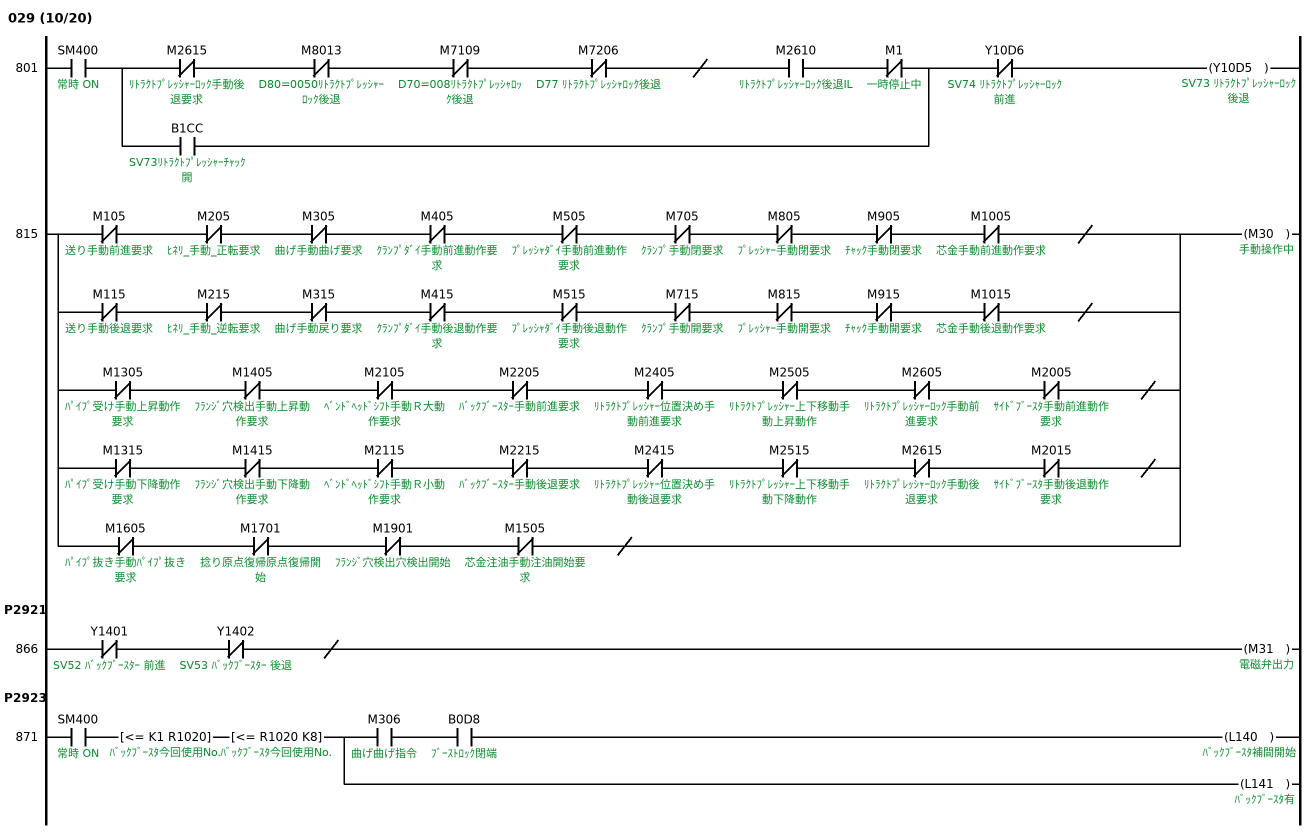
801   LD      SM400  ; 常時 ON
      LDI     M2615  ; ﾘﾄﾗｸﾄﾌﾟﾚｯｼｬｰﾛｯｸ手動後退要求
      ANI     M8013  ; D80=0050ﾘﾄﾗｸﾄﾌﾟﾚｯｼｬｰﾛｯｸ後退
      ANI     M7109  ; D70=008ﾘﾄﾗｸﾄﾌﾟﾚｯｼｬﾛｯｸ後退
      ANI     M7206  ; D77 ﾘﾄﾗｸﾄﾌﾟﾚｯｼｬﾛｯｸ後退
      INV
      AND     M2610  ; ﾘﾄﾗｸﾄﾌﾟﾚｯｼｬｰﾛｯｸ後退IL
      ANI     M1  ; 一時停止中
      OR      B1CC  ; SV73ﾘﾄﾗｸﾄﾌﾟﾚｯｼｬｰﾁｬｯｸ 開
      ANB
      ANI     Y10D6  ; SV74 ﾘﾄﾗｸﾄﾌﾟﾚｯｼｬｰﾛｯｸ 前進
      OUT     Y10D5  ; SV73 ﾘﾄﾗｸﾄﾌﾟﾚｯｼｬｰﾛｯｸ 後退
; 
815   LDI     M105  ; 送り手動前進要求
      ANI     M205  ; ﾋﾈﾘ_手動_正転要求
      ANI     M305  ; 曲げ手動曲げ要求
      ANI     M405  ; ｸﾗﾝﾌﾟﾀﾞｲ手動前進動作要求
      ANI     M505  ; ﾌﾟﾚｯｼｬﾀﾞｲ手動前進動作要求
      ANI     M705  ; ｸﾗﾝﾌﾟ手動閉要求
      ANI     M805  ; ﾌﾟﾚｯｼｬｰ手動閉要求
      ANI     M905  ; ﾁｬｯｸ手動閉要求
      ANI     M1005  ; 芯金手動前進動作要求
      INV
      LDI     M115  ; 送り手動後退要求
      ANI     M215  ; ﾋﾈﾘ_手動_逆転要求
      ANI     M315  ; 曲げ手動戻り要求
      ANI     M415  ; ｸﾗﾝﾌﾟﾀﾞｲ手動後退動作要求
      ANI     M515  ; ﾌﾟﾚｯｼｬﾀﾞｲ手動後退動作要求
      ANI     M715  ; ｸﾗﾝﾌﾟ手動開要求
      ANI     M815  ; ﾌﾟﾚｯｼｬｰ手動開要求
      ANI     M915  ; ﾁｬｯｸ手動開要求
      ANI     M1015  ; 芯金手動後退動作要求
      INV
      ORB
      LDI     M1305  ; ﾊﾟｲﾌﾟ受け手動上昇動作要求
      ANI     M1405  ; ﾌﾗﾝｼﾞ穴検出手動上昇動作要求
      ANI     M2105  ; ﾍﾞﾝﾄﾞﾍｯﾄﾞｼﾌﾄ手動Ｒ大動作要求
      ANI     M2205  ; ﾊﾞｯｸﾌﾞｰｽﾀｰ手動前進要求
      ANI     M2405  ; ﾘﾄﾗｸﾄﾌﾟﾚｯｼｬｰ位置決め手動前進要求
      ANI     M2505  ; ﾘﾄﾗｸﾄﾌﾟﾚｯｼｬｰ上下移動手動上昇動作
      ANI     M2605  ; ﾘﾄﾗｸﾄﾌﾟﾚｯｼｬｰﾛｯｸ手動前進要求
      ANI     M2005  ; ｻｲﾄﾞﾌﾞｰｽﾀ手動前進動作要求
      INV
      ORB
      LDI     M1315  ; ﾊﾟｲﾌﾟ受け手動下降動作要求
      ANI     M1415  ; ﾌﾗﾝｼﾞ穴検出手動下降動作要求
      ANI     M2115  ; ﾍﾞﾝﾄﾞﾍｯﾄﾞｼﾌﾄ手動Ｒ小動作要求
      ANI     M2215  ; ﾊﾞｯｸﾌﾞｰｽﾀｰ手動後退要求
      ANI     M2415  ; ﾘﾄﾗｸﾄﾌﾟﾚｯｼｬｰ位置決め手動後退要求
      ANI     M2515  ; ﾘﾄﾗｸﾄﾌﾟﾚｯｼｬｰ上下移動手動下降動作
      ANI     M2615  ; ﾘﾄﾗｸﾄﾌﾟﾚｯｼｬｰﾛｯｸ手動後退要求
      ANI     M2015  ; ｻｲﾄﾞﾌﾞｰｽﾀ手動後退動作要求
      INV
      ORB
      LDI     M1605  ; ﾊﾟｲﾌﾟ抜き手動ﾊﾟｲﾌﾟ抜き要求
      ANI     M1701  ; 捻り原点復帰原点復帰開始
      ANI     M1901  ; ﾌﾗﾝｼﾞ穴検出穴検出開始
      ANI     M1505  ; 芯金注油手動注油開始要求
      INV
      ORB
      OUT     M30  ; 手動操作中
; 
      P2921
866   LDI     Y1401  ; SV52 ﾊﾞｯｸﾌﾞｰｽﾀｰ 前進
      ANI     Y1402  ; SV53 ﾊﾞｯｸﾌﾞｰｽﾀｰ 後退
      INV
      OUT     M31  ; 電磁弁出力
      P2923
871   LD      SM400  ; 常時 ON
      AND<=   K1 R1020  ; ﾊﾞｯｸﾌﾞｰｽﾀ今回使用No.
      AND<=   R1020 K8  ; ﾊﾞｯｸﾌﾞｰｽﾀ今回使用No.
      MPS
      AND     M306  ; 曲げ曲げ指令
      AND     B0D8  ; ﾌﾞｰｽﾄﾛｯｸ閉端
      OUT     L140  ; ﾊﾞｯｸﾌﾞｰｽﾀ補間開始
      MPP
      OUT     L141  ; ﾊﾞｯｸﾌﾞｰｽﾀ有
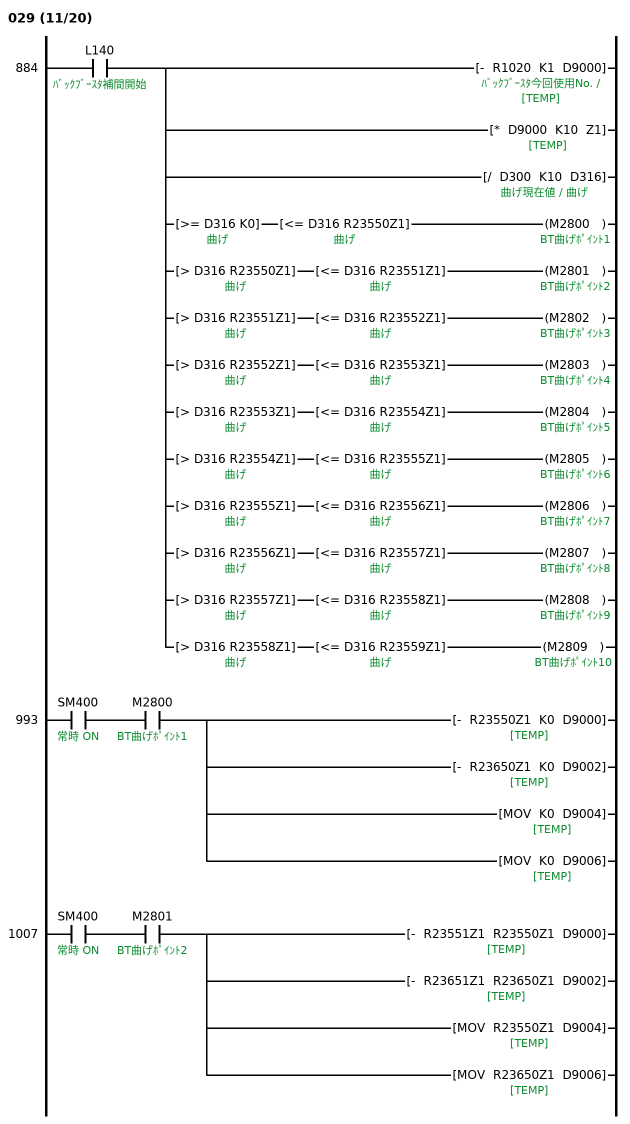
884   LD      L140  ; ﾊﾞｯｸﾌﾞｰｽﾀ補間開始
      -       R1020 K1 D9000  ; [TEMP]
      *       D9000 K10 Z1
      /       D300 K10 D316  ; 曲げ現在値 / 曲げ
      MPS
      AND>=   D316 K0  ; 曲げ
      AND<=   D316 R23550Z1  ; 曲げ
      OUT     M2800  ; BT曲げﾎﾟｲﾝﾄ1
      MRD
      AND>    D316 R23550Z1  ; 曲げ
      AND<=   D316 R23551Z1  ; 曲げ
      OUT     M2801  ; BT曲げﾎﾟｲﾝﾄ2
      MRD
      AND>    D316 R23551Z1  ; 曲げ
      AND<=   D316 R23552Z1  ; 曲げ
      OUT     M2802  ; BT曲げﾎﾟｲﾝﾄ3
      MRD
      AND>    D316 R23552Z1  ; 曲げ
      AND<=   D316 R23553Z1  ; 曲げ
      OUT     M2803  ; BT曲げﾎﾟｲﾝﾄ4
      MRD
      AND>    D316 R23553Z1  ; 曲げ
      AND<=   D316 R23554Z1  ; 曲げ
      OUT     M2804  ; BT曲げﾎﾟｲﾝﾄ5
      MRD
      AND>    D316 R23554Z1  ; 曲げ
      AND<=   D316 R23555Z1  ; 曲げ
      OUT     M2805  ; BT曲げﾎﾟｲﾝﾄ6
      MRD
      AND>    D316 R23555Z1  ; 曲げ
      AND<=   D316 R23556Z1  ; 曲げ
      OUT     M2806  ; BT曲げﾎﾟｲﾝﾄ7
      MRD
      AND>    D316 R23556Z1  ; 曲げ
      AND<=   D316 R23557Z1  ; 曲げ
      OUT     M2807  ; BT曲げﾎﾟｲﾝﾄ8
      MRD
      AND>    D316 R23557Z1  ; 曲げ
      AND<=   D316 R23558Z1  ; 曲げ
      OUT     M2808  ; BT曲げﾎﾟｲﾝﾄ9
      MPP
      AND>    D316 R23558Z1  ; 曲げ
      AND<=   D316 R23559Z1  ; 曲げ
      OUT     M2809  ; BT曲げﾎﾟｲﾝﾄ10
993   LD      SM400  ; 常時 ON
      AND     M2800  ; BT曲げﾎﾟｲﾝﾄ1
      -       R23550Z1 K0 D9000
      -       R23650Z1 K0 D9002  ; [TEMP]
      MOV     K0 D9004  ; [TEMP]
      MOV     K0 D9006  ; [TEMP]
1007  LD      SM400  ; 常時 ON
      AND     M2801  ; BT曲げﾎﾟｲﾝﾄ2
      -       R23551Z1 R23550Z1 D9000
      -       R23651Z1 R23650Z1 D9002
      MOV     R23550Z1 D9004
      MOV     R23650Z1 D9006
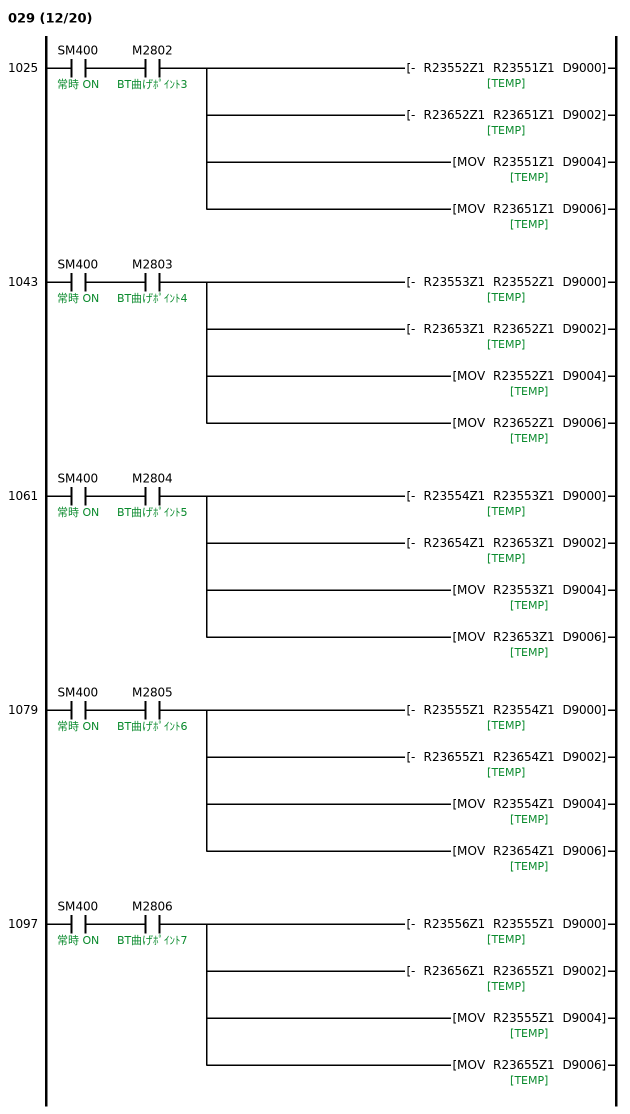
1025  LD      SM400  ; 常時 ON
      AND     M2802  ; BT曲げﾎﾟｲﾝﾄ3
      -       R23552Z1 R23551Z1 D9000
      -       R23652Z1 R23651Z1 D9002
      MOV     R23551Z1 D9004
      MOV     R23651Z1 D9006
1043  LD      SM400  ; 常時 ON
      AND     M2803  ; BT曲げﾎﾟｲﾝﾄ4
      -       R23553Z1 R23552Z1 D9000
      -       R23653Z1 R23652Z1 D9002
      MOV     R23552Z1 D9004
      MOV     R23652Z1 D9006
1061  LD      SM400  ; 常時 ON
      AND     M2804  ; BT曲げﾎﾟｲﾝﾄ5
      -       R23554Z1 R23553Z1 D9000
      -       R23654Z1 R23653Z1 D9002
      MOV     R23553Z1 D9004
      MOV     R23653Z1 D9006
1079  LD      SM400  ; 常時 ON
      AND     M2805  ; BT曲げﾎﾟｲﾝﾄ6
      -       R23555Z1 R23554Z1 D9000
      -       R23655Z1 R23654Z1 D9002
      MOV     R23554Z1 D9004
      MOV     R23654Z1 D9006
1097  LD      SM400  ; 常時 ON
      AND     M2806  ; BT曲げﾎﾟｲﾝﾄ7
      -       R23556Z1 R23555Z1 D9000
      -       R23656Z1 R23655Z1 D9002
      MOV     R23555Z1 D9004
      MOV     R23655Z1 D9006
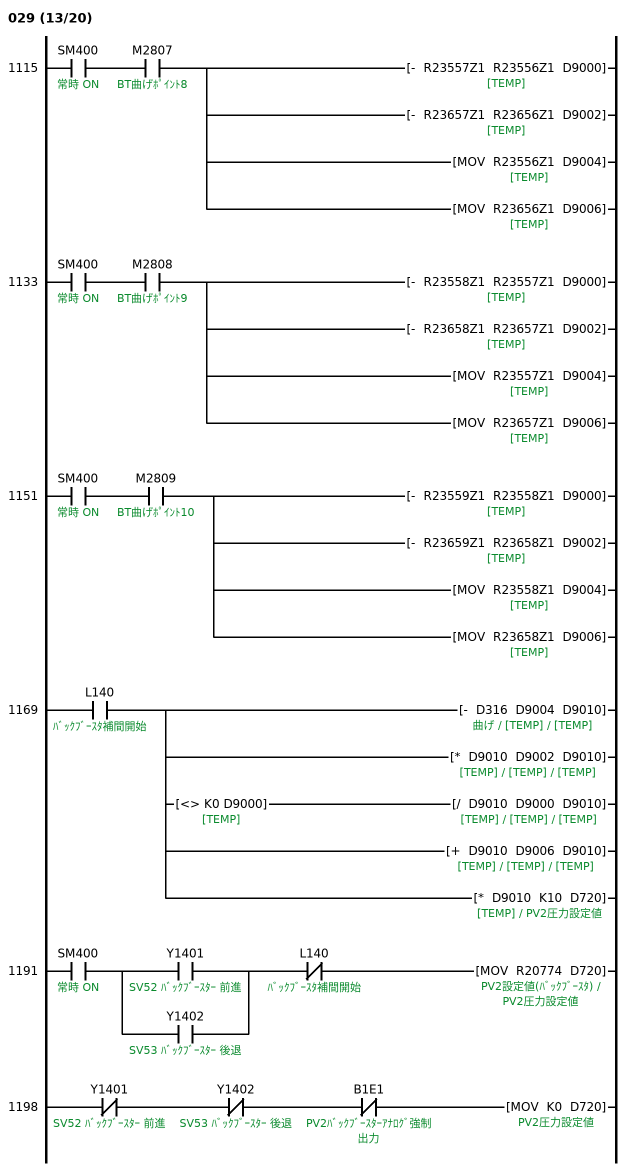
1115  LD      SM400  ; 常時 ON
      AND     M2807  ; BT曲げﾎﾟｲﾝﾄ8
      -       R23557Z1 R23556Z1 D9000
      -       R23657Z1 R23656Z1 D9002
      MOV     R23556Z1 D9004
      MOV     R23656Z1 D9006
1133  LD      SM400  ; 常時 ON
      AND     M2808  ; BT曲げﾎﾟｲﾝﾄ9
      -       R23558Z1 R23557Z1 D9000
      -       R23658Z1 R23657Z1 D9002
      MOV     R23557Z1 D9004
      MOV     R23657Z1 D9006
1151  LD      SM400  ; 常時 ON
      AND     M2809  ; BT曲げﾎﾟｲﾝﾄ10
      -       R23559Z1 R23558Z1 D9000
      -       R23659Z1 R23658Z1 D9002
      MOV     R23558Z1 D9004
      MOV     R23658Z1 D9006
1169  LD      L140  ; ﾊﾞｯｸﾌﾞｰｽﾀ補間開始
      -       D316 D9004 D9010  ; [TEMP]
      *       D9010 D9002 D9010
      MPS
      AND<>   K0 D9000  ; [TEMP]
      /       D9010 D9000 D9010
      MPP
      +       D9010 D9006 D9010
      *       D9010 K10 D720  ; PV2圧力設定値
1191  LD      SM400  ; 常時 ON
      LD      Y1401  ; SV52 ﾊﾞｯｸﾌﾞｰｽﾀｰ 前進
      OR      Y1402  ; SV53 ﾊﾞｯｸﾌﾞｰｽﾀｰ 後退
      ANB
      ANI     L140  ; ﾊﾞｯｸﾌﾞｰｽﾀ補間開始
      MOV     R20774 D720  ; PV2設定値(ﾊﾞｯｸﾌﾞｰｽﾀ)
1198  LDI     Y1401  ; SV52 ﾊﾞｯｸﾌﾞｰｽﾀｰ 前進
      ANI     Y1402  ; SV53 ﾊﾞｯｸﾌﾞｰｽﾀｰ 後退
      ANI     B1E1  ; PV2ﾊﾞｯｸﾌﾞｰｽﾀｰｱﾅﾛｸﾞ強制出力
      MOV     K0 D720
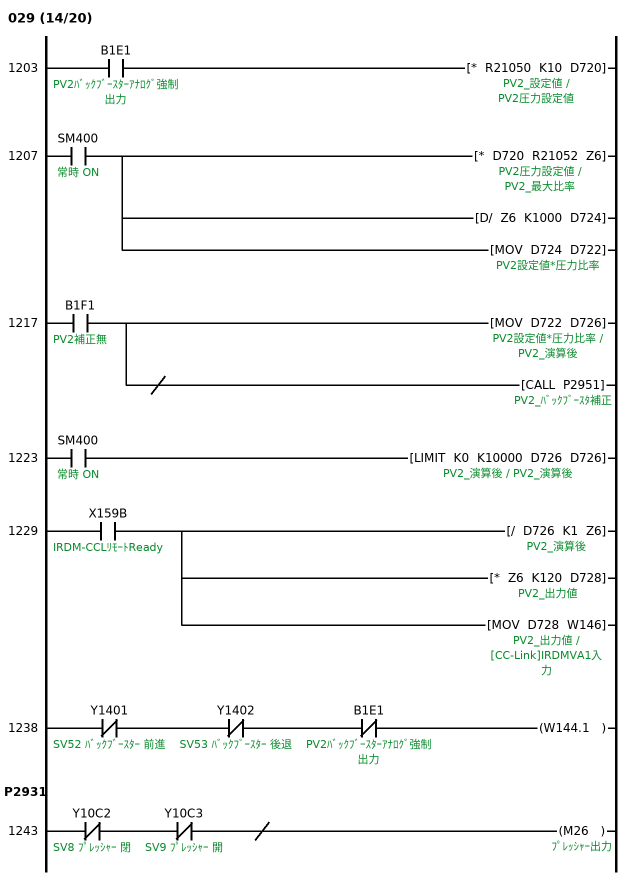
1203  LD      B1E1  ; PV2ﾊﾞｯｸﾌﾞｰｽﾀｰｱﾅﾛｸﾞ強制出力
      *       R21050 K10 D720  ; PV2_設定値
1207  LD      SM400  ; 常時 ON
      *       D720 R21052 Z6  ; PV2_最大比率
      D/      Z6 K1000 D724
      MOV     D724 D722  ; PV2設定値*圧力比率
1217  LD      B1F1  ; PV2補正無
      MOV     D722 D726  ; PV2_演算後
      INV
      CALL    P2951  ; PV2_ﾊﾞｯｸﾌﾞｰｽﾀ補正
1223  LD      SM400  ; 常時 ON
      LIMIT   K0 K10000 D726 D726
1229  LD      X159B  ; IRDM-CCLﾘﾓｰﾄReady
      /       D726 K1 Z6
      *       Z6 K120 D728  ; PV2_出力値
      MOV     D728 W146  ; [CC-Link]IRDMVA1入力
1238  LDI     Y1401  ; SV52 ﾊﾞｯｸﾌﾞｰｽﾀｰ 前進
      ANI     Y1402  ; SV53 ﾊﾞｯｸﾌﾞｰｽﾀｰ 後退
      ANI     B1E1  ; PV2ﾊﾞｯｸﾌﾞｰｽﾀｰｱﾅﾛｸﾞ強制出力
      OUT     W144.1
      P2931
1243  LDI     Y10C2  ; SV8 ﾌﾟﾚｯｼｬｰ 閉
      ANI     Y10C3  ; SV9 ﾌﾟﾚｯｼｬｰ 開
      INV
      OUT     M26  ; ﾌﾟﾚｯｼｬｰ出力
      P2932
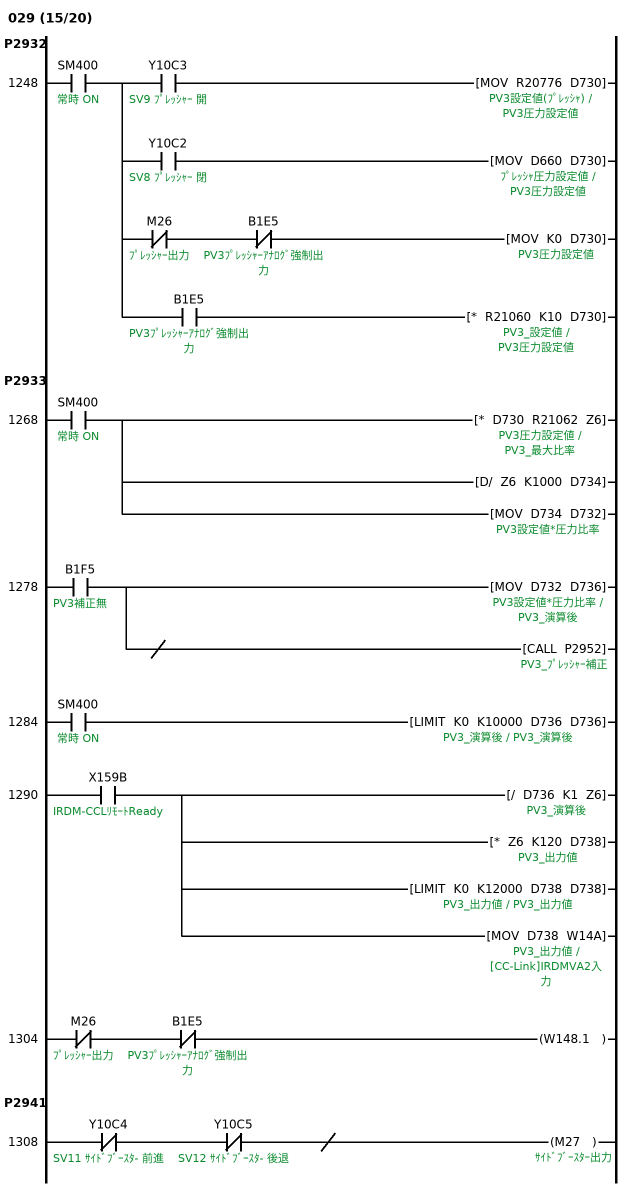
1248  LD      SM400  ; 常時 ON
      MPS
      AND     Y10C3  ; SV9 ﾌﾟﾚｯｼｬｰ 開
      MOV     R20776 D730  ; PV3設定値(ﾌﾟﾚｯｼｬ) / PV3圧力設定値
      MRD
      AND     Y10C2  ; SV8 ﾌﾟﾚｯｼｬｰ 閉
      MOV     D660 D730  ; ﾌﾟﾚｯｼｬ圧力設定値
      MRD
      ANI     M26  ; ﾌﾟﾚｯｼｬｰ出力
      ANI     B1E5  ; PV3ﾌﾟﾚｯｼｬｰｱﾅﾛｸﾞ強制出力
      MOV     K0 D730
      MPP
      AND     B1E5  ; PV3ﾌﾟﾚｯｼｬｰｱﾅﾛｸﾞ強制出力
      *       R21060 K10 D730  ; PV3_設定値
      P2933
1268  LD      SM400  ; 常時 ON
      *       D730 R21062 Z6  ; PV3_最大比率
      D/      Z6 K1000 D734
      MOV     D734 D732  ; PV3設定値*圧力比率
1278  LD      B1F5  ; PV3補正無
      MOV     D732 D736  ; PV3_演算後
      INV
      CALL    P2952  ; PV3_ﾌﾟﾚｯｼｬｰ補正
1284  LD      SM400  ; 常時 ON
      LIMIT   K0 K10000 D736 D736
1290  LD      X159B  ; IRDM-CCLﾘﾓｰﾄReady
      /       D736 K1 Z6
      *       Z6 K120 D738  ; PV3_出力値
      LIMIT   K0 K12000 D738 D738
      MOV     D738 W14A  ; [CC-Link]IRDMVA2入力
1304  LDI     M26  ; ﾌﾟﾚｯｼｬｰ出力
      ANI     B1E5  ; PV3ﾌﾟﾚｯｼｬｰｱﾅﾛｸﾞ強制出力
      OUT     W148.1
      P2941
1308  LDI     Y10C4  ; SV11 ｻｲﾄﾞﾌﾞｰｽﾀ- 前進
      ANI     Y10C5  ; SV12 ｻｲﾄﾞﾌﾞｰｽﾀ- 後退
      INV
      OUT     M27  ; ｻｲﾄﾞﾌﾞｰｽﾀｰ出力
      P2942
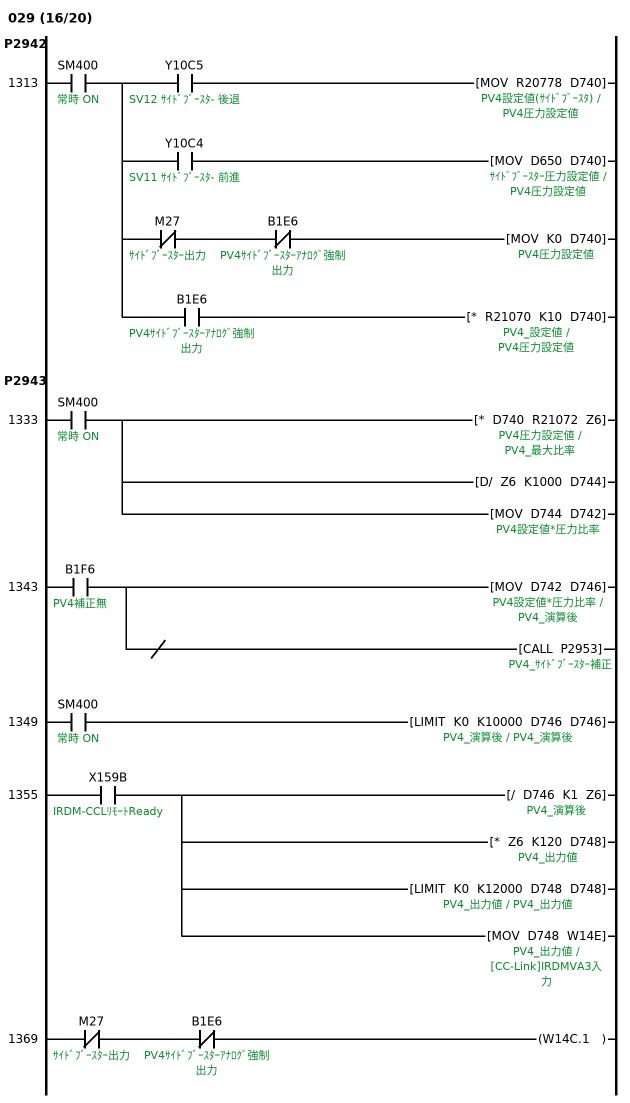
1313  LD      SM400  ; 常時 ON
      MPS
      AND     Y10C5  ; SV12 ｻｲﾄﾞﾌﾞｰｽﾀ- 後退
      MOV     R20778 D740  ; PV4設定値(ｻｲﾄﾞﾌﾞｰｽﾀ) / PV4圧力設定値
      MRD
      AND     Y10C4  ; SV11 ｻｲﾄﾞﾌﾞｰｽﾀ- 前進
      MOV     D650 D740  ; ｻｲﾄﾞﾌﾞｰｽﾀｰ圧力設定値
      MRD
      ANI     M27  ; ｻｲﾄﾞﾌﾞｰｽﾀｰ出力
      ANI     B1E6  ; PV4ｻｲﾄﾞﾌﾞｰｽﾀｰｱﾅﾛｸﾞ強制出力
      MOV     K0 D740
      MPP
      AND     B1E6  ; PV4ｻｲﾄﾞﾌﾞｰｽﾀｰｱﾅﾛｸﾞ強制出力
      *       R21070 K10 D740  ; PV4_設定値
      P2943
1333  LD      SM400  ; 常時 ON
      *       D740 R21072 Z6  ; PV4_最大比率
      D/      Z6 K1000 D744
      MOV     D744 D742  ; PV4設定値*圧力比率
1343  LD      B1F6  ; PV4補正無
      MOV     D742 D746  ; PV4_演算後
      INV
      CALL    P2953  ; PV4_ｻｲﾄﾞﾌﾞｰｽﾀｰ補正
1349  LD      SM400  ; 常時 ON
      LIMIT   K0 K10000 D746 D746
1355  LD      X159B  ; IRDM-CCLﾘﾓｰﾄReady
      /       D746 K1 Z6
      *       Z6 K120 D748  ; PV4_出力値
      LIMIT   K0 K12000 D748 D748
      MOV     D748 W14E  ; [CC-Link]IRDMVA3入力
1369  LDI     M27  ; ｻｲﾄﾞﾌﾞｰｽﾀｰ出力
      ANI     B1E6  ; PV4ｻｲﾄﾞﾌﾞｰｽﾀｰｱﾅﾛｸﾞ強制出力
      OUT     W14C.1
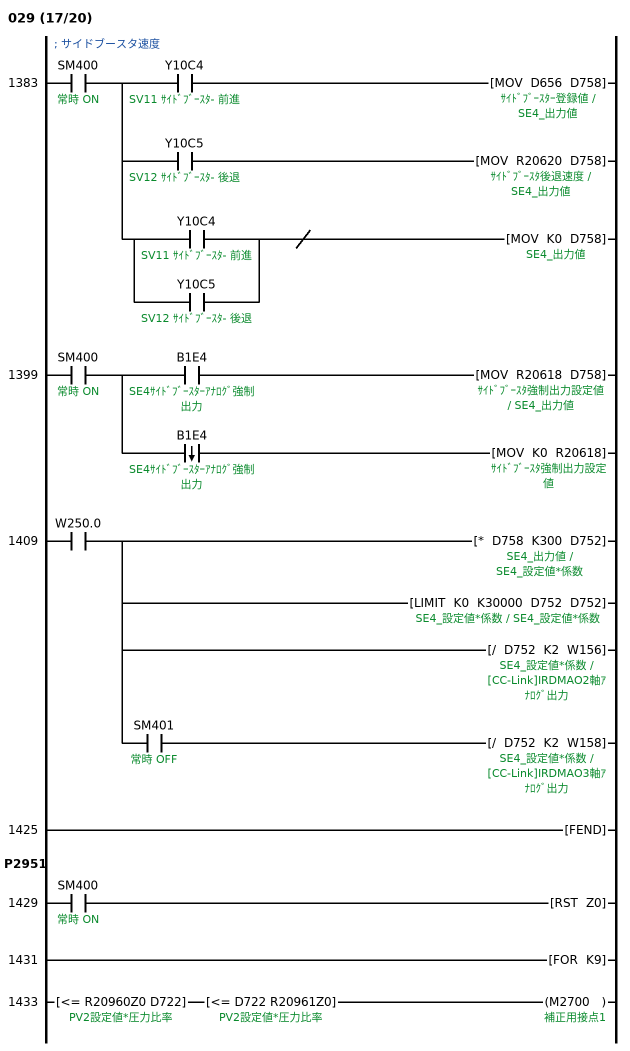
; サイドブースタ速度
1383  LD      SM400  ; 常時 ON
      MPS
      AND     Y10C4  ; SV11 ｻｲﾄﾞﾌﾞｰｽﾀ- 前進
      MOV     D656 D758  ; ｻｲﾄﾞﾌﾞｰｽﾀｰ登録値 / SE4_出力値
      MRD
      AND     Y10C5  ; SV12 ｻｲﾄﾞﾌﾞｰｽﾀ- 後退
      MOV     R20620 D758  ; ｻｲﾄﾞﾌﾞｰｽﾀ後退速度
      MPP
      LD      Y10C4  ; SV11 ｻｲﾄﾞﾌﾞｰｽﾀ- 前進
      OR      Y10C5  ; SV12 ｻｲﾄﾞﾌﾞｰｽﾀ- 後退
      ANB
      INV
      MOV     K0 D758
1399  LD      SM400  ; 常時 ON
      MPS
      AND     B1E4  ; SE4ｻｲﾄﾞﾌﾞｰｽﾀｰｱﾅﾛｸﾞ強制出力
      MOV     R20618 D758  ; ｻｲﾄﾞﾌﾞｰｽﾀ強制出力設定値
      MPP
      ANDF    B1E4  ; SE4ｻｲﾄﾞﾌﾞｰｽﾀｰｱﾅﾛｸﾞ強制出力
      MOV     K0 R20618
1409  LD      W250.0
      *       D758 K300 D752  ; SE4_設定値*係数
      LIMIT   K0 K30000 D752 D752
      /       D752 K2 W156  ; [CC-Link]IRDMAO2軸ｱﾅﾛｸﾞ出力
      AND     SM401  ; 常時 OFF
      /       D752 K2 W158  ; [CC-Link]IRDMAO3軸ｱﾅﾛｸﾞ出力
1425  FEND
; 
      P2951
1429  LD      SM400  ; 常時 ON
      RST     Z0
1431  FOR     K9
1433  LD<=    R20960Z0 D722  ; PV2設定値*圧力比率
      AND<=   D722 R20961Z0  ; PV2設定値*圧力比率
      OUT     M2700  ; 補正用接点1
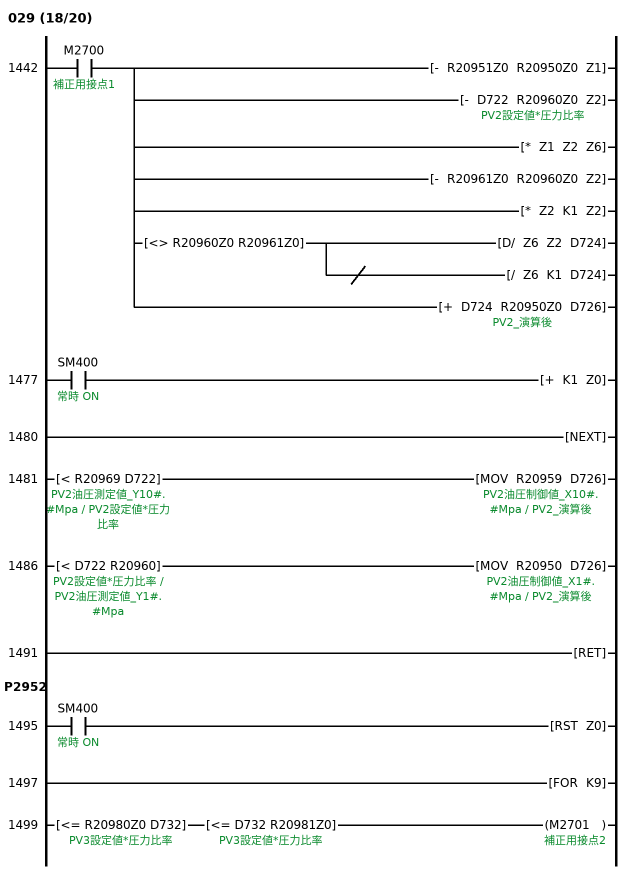
1442  LD      M2700  ; 補正用接点1
      -       R20951Z0 R20950Z0 Z1
      -       D722 R20960Z0 Z2
      *       Z1 Z2 Z6
      -       R20961Z0 R20960Z0 Z2
      *       Z2 K1 Z2
      MPS
      AND<>   R20960Z0 R20961Z0
      D/      Z6 Z2 D724
      INV
      /       Z6 K1 D724
      MPP
      +       D724 R20950Z0 D726
1477  LD      SM400  ; 常時 ON
      +       K1 Z0
1480  NEXT
1481  LD<     R20969 D722  ; PV2油圧測定値_Y10#.#Mpa / PV2設定値*圧力比率
      MOV     R20959 D726  ; PV2油圧制御値_X10#.#Mpa
1486  LD<     D722 R20960  ; PV2設定値*圧力比率 / PV2油圧測定値_Y1#.#Mpa
      MOV     R20950 D726  ; PV2油圧制御値_X1#.#Mpa
1491  RET
; 
      P2952
1495  LD      SM400  ; 常時 ON
      RST     Z0
1497  FOR     K9
1499  LD<=    R20980Z0 D732  ; PV3設定値*圧力比率
      AND<=   D732 R20981Z0  ; PV3設定値*圧力比率
      OUT     M2701  ; 補正用接点2
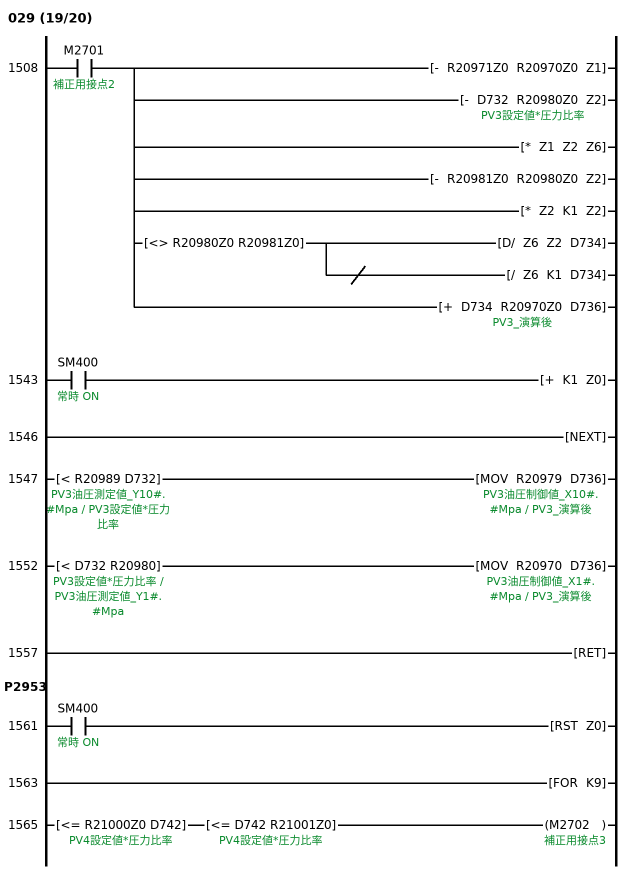
1508  LD      M2701  ; 補正用接点2
      -       R20971Z0 R20970Z0 Z1
      -       D732 R20980Z0 Z2
      *       Z1 Z2 Z6
      -       R20981Z0 R20980Z0 Z2
      *       Z2 K1 Z2
      MPS
      AND<>   R20980Z0 R20981Z0
      D/      Z6 Z2 D734
      INV
      /       Z6 K1 D734
      MPP
      +       D734 R20970Z0 D736
1543  LD      SM400  ; 常時 ON
      +       K1 Z0
1546  NEXT
1547  LD<     R20989 D732  ; PV3油圧測定値_Y10#.#Mpa / PV3設定値*圧力比率
      MOV     R20979 D736  ; PV3油圧制御値_X10#.#Mpa
1552  LD<     D732 R20980  ; PV3設定値*圧力比率 / PV3油圧測定値_Y1#.#Mpa
      MOV     R20970 D736  ; PV3油圧制御値_X1#.#Mpa
1557  RET
; 
      P2953
1561  LD      SM400  ; 常時 ON
      RST     Z0
1563  FOR     K9
1565  LD<=    R21000Z0 D742  ; PV4設定値*圧力比率
      AND<=   D742 R21001Z0  ; PV4設定値*圧力比率
      OUT     M2702  ; 補正用接点3
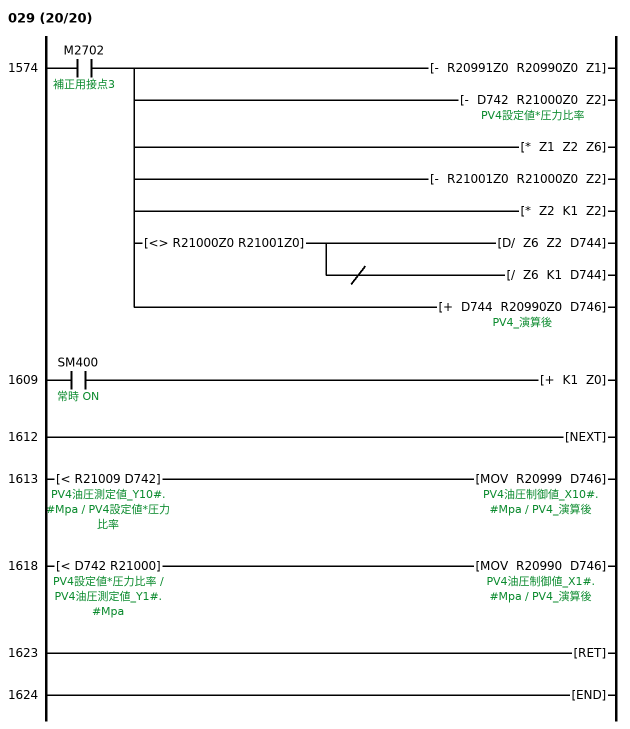
1574  LD      M2702  ; 補正用接点3
      -       R20991Z0 R20990Z0 Z1
      -       D742 R21000Z0 Z2
      *       Z1 Z2 Z6
      -       R21001Z0 R21000Z0 Z2
      *       Z2 K1 Z2
      MPS
      AND<>   R21000Z0 R21001Z0
      D/      Z6 Z2 D744
      INV
      /       Z6 K1 D744
      MPP
      +       D744 R20990Z0 D746
1609  LD      SM400  ; 常時 ON
      +       K1 Z0
1612  NEXT
1613  LD<     R21009 D742  ; PV4油圧測定値_Y10#.#Mpa / PV4設定値*圧力比率
      MOV     R20999 D746  ; PV4油圧制御値_X10#.#Mpa
1618  LD<     D742 R21000  ; PV4設定値*圧力比率 / PV4油圧測定値_Y1#.#Mpa
      MOV     R20990 D746  ; PV4油圧制御値_X1#.#Mpa
1623  RET
1624  END
END_PROGRAM

PROGRAM 030  // TP&表示
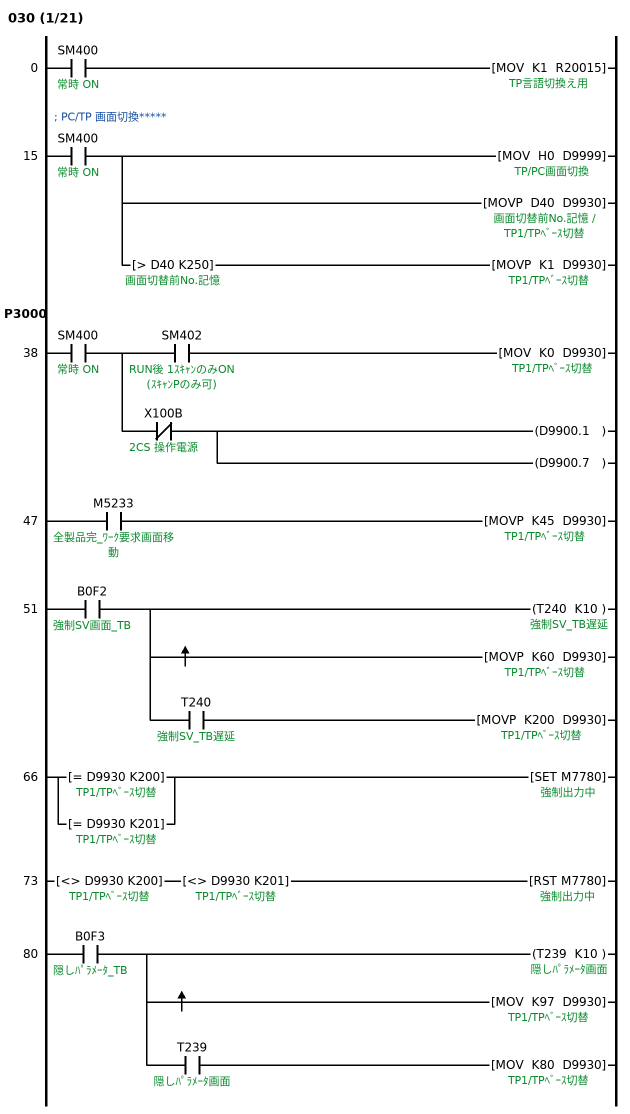
0     LD      SM400  ; 常時 ON
      MOV     K1 R20015  ; TP言語切換え用
; PC/TP 画面切換*****
15    LD      SM400  ; 常時 ON
      MOV     H0 D9999  ; TP/PC画面切換
        [note] ﾀｯﾁﾊﾟﾈﾙ画面
      MOVP    D40 D9930  ; 画面切替前No.記憶 / TP1/TPﾍﾞｰｽ切替
      AND>    D40 K250  ; 画面切替前No.記憶
      MOVP    K1 D9930
; 
      P3000
38    LD      SM400  ; 常時 ON
      MPS
      AND     SM402  ; RUN後 1ｽｷｬﾝのみON (ｽｷｬﾝPのみ可)
      MOV     K0 D9930
      MPP
      ANI     X100B  ; 2CS 操作電源
      OUT     D9900.1
      OUT     D9900.7
47    LD      M5233  ; 全製品完_ﾜｰｸ要求画面移動
      MOVP    K45 D9930
51    LD      B0F2  ; 強制SV画面_TB
      OUT     T240 K10  ; 強制SV_TB遅延
      MPS
      MEP
      MOVP    K60 D9930
      MPP
      AND     T240  ; 強制SV_TB遅延
      MOVP    K200 D9930
66    LD=     D9930 K200  ; TP1/TPﾍﾞｰｽ切替
      OR=     D9930 K201  ; TP1/TPﾍﾞｰｽ切替
      SET     M7780  ; 強制出力中
73    LD<>    D9930 K200  ; TP1/TPﾍﾞｰｽ切替
      AND<>   D9930 K201  ; TP1/TPﾍﾞｰｽ切替
      RST     M7780  ; 強制出力中
80    LD      B0F3  ; 隠しﾊﾟﾗﾒｰﾀ_TB
      OUT     T239 K10  ; 隠しﾊﾟﾗﾒｰﾀ画面
      MPS
      MEP
      MOV     K97 D9930
      MPP
      AND     T239  ; 隠しﾊﾟﾗﾒｰﾀ画面
      MOV     K80 D9930
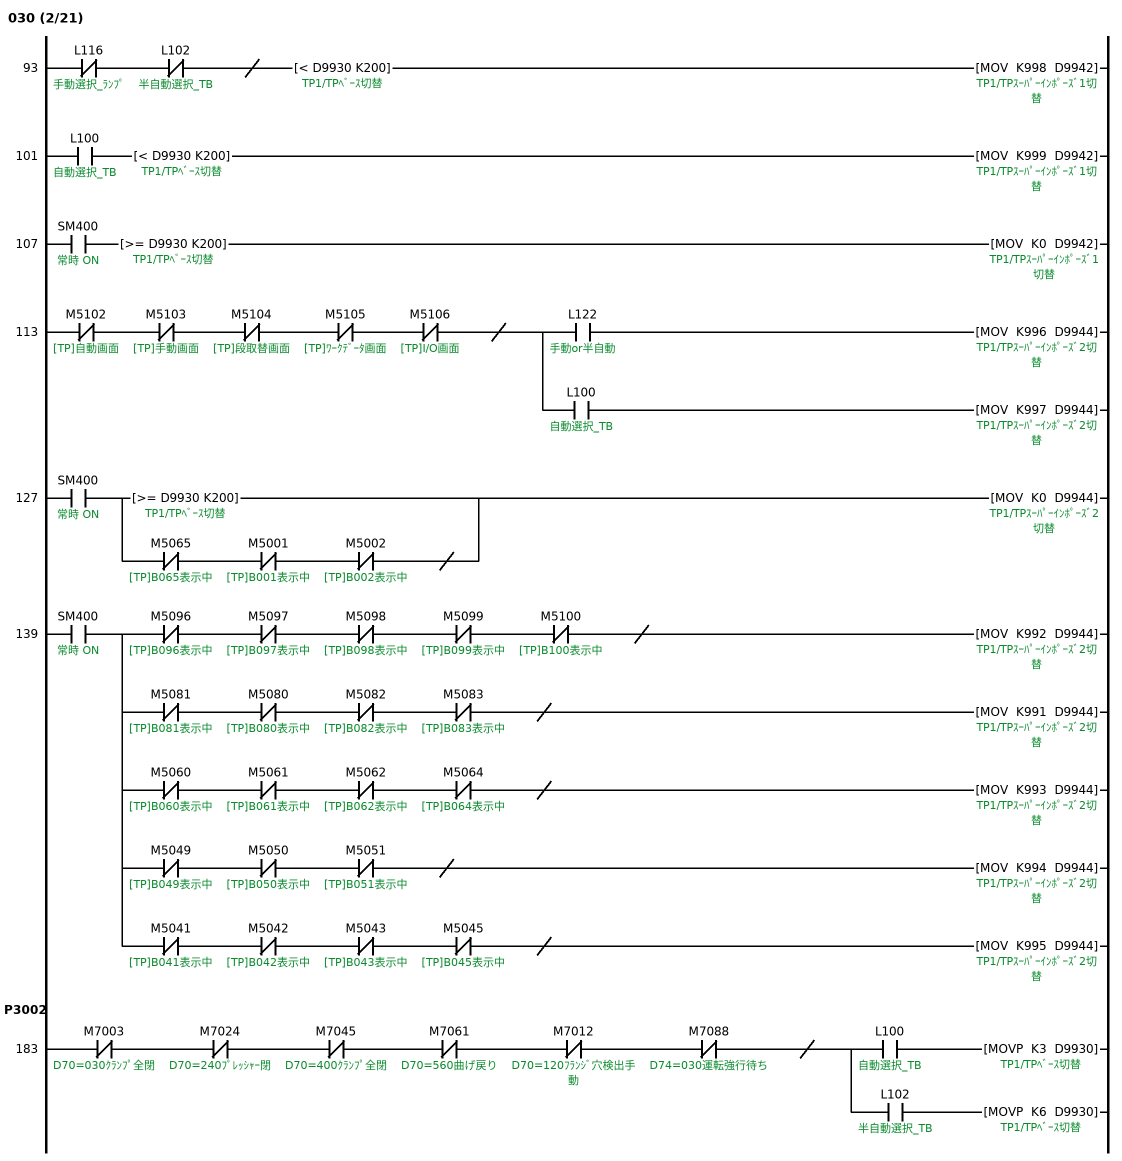
93    LDI     L116  ; 手動選択_ﾗﾝﾌﾟ
      ANI     L102  ; 半自動選択_TB
      INV
      AND<    D9930 K200  ; TP1/TPﾍﾞｰｽ切替
      MOV     K998 D9942  ; TP1/TPｽｰﾊﾟｰｲﾝﾎﾟｰｽﾞ1切替
101   LD      L100  ; 自動選択_TB
      AND<    D9930 K200  ; TP1/TPﾍﾞｰｽ切替
      MOV     K999 D9942
107   LD      SM400  ; 常時 ON
      AND>=   D9930 K200  ; TP1/TPﾍﾞｰｽ切替
      MOV     K0 D9942
113   LDI     M5102  ; [TP]自動画面
      ANI     M5103  ; [TP]手動画面
      ANI     M5104  ; [TP]段取替画面
      ANI     M5105  ; [TP]ﾜｰｸﾃﾞｰﾀ画面
      ANI     M5106  ; [TP]I/O画面
      INV
      MPS
      AND     L122  ; 手動or半自動
      MOV     K996 D9944  ; TP1/TPｽｰﾊﾟｰｲﾝﾎﾟｰｽﾞ2切替
      MPP
      AND     L100  ; 自動選択_TB
      MOV     K997 D9944
127   LD      SM400  ; 常時 ON
      LD>=    D9930 K200  ; TP1/TPﾍﾞｰｽ切替
      LDI     M5065  ; [TP]B065表示中
      ANI     M5001  ; [TP]B001表示中
      ANI     M5002  ; [TP]B002表示中
      INV
      ORB
      ANB
      MOV     K0 D9944
139   LD      SM400  ; 常時 ON
      MPS
      ANI     M5096  ; [TP]B096表示中
      ANI     M5097  ; [TP]B097表示中
      ANI     M5098  ; [TP]B098表示中
      ANI     M5099  ; [TP]B099表示中
      ANI     M5100  ; [TP]B100表示中
      INV
      MOV     K992 D9944
      MRD
      ANI     M5081  ; [TP]B081表示中
      ANI     M5080  ; [TP]B080表示中
      ANI     M5082  ; [TP]B082表示中
      ANI     M5083  ; [TP]B083表示中
      INV
      MOV     K991 D9944
      MRD
      ANI     M5060  ; [TP]B060表示中
      ANI     M5061  ; [TP]B061表示中
      ANI     M5062  ; [TP]B062表示中
      ANI     M5064  ; [TP]B064表示中
      INV
      MOV     K993 D9944
      MRD
      ANI     M5049  ; [TP]B049表示中
      ANI     M5050  ; [TP]B050表示中
      ANI     M5051  ; [TP]B051表示中
      INV
      MOV     K994 D9944
      MPP
      ANI     M5041  ; [TP]B041表示中
      ANI     M5042  ; [TP]B042表示中
      ANI     M5043  ; [TP]B043表示中
      ANI     M5045  ; [TP]B045表示中
      INV
      MOV     K995 D9944
; 
      P3002
183   LDI     M7003  ; D70=030ｸﾗﾝﾌﾟ全閉
      ANI     M7024  ; D70=240ﾌﾟﾚｯｼｬｰ閉
      ANI     M7045  ; D70=400ｸﾗﾝﾌﾟ全閉
      ANI     M7061  ; D70=560曲げ戻り
      ANI     M7012  ; D70=120ﾌﾗﾝｼﾞ穴検出手動
      ANI     M7088  ; D74=030運転強行待ち
      INV
      MPS
      AND     L100  ; 自動選択_TB
      MOVP    K3 D9930
      MPP
      AND     L102  ; 半自動選択_TB
      MOVP    K6 D9930
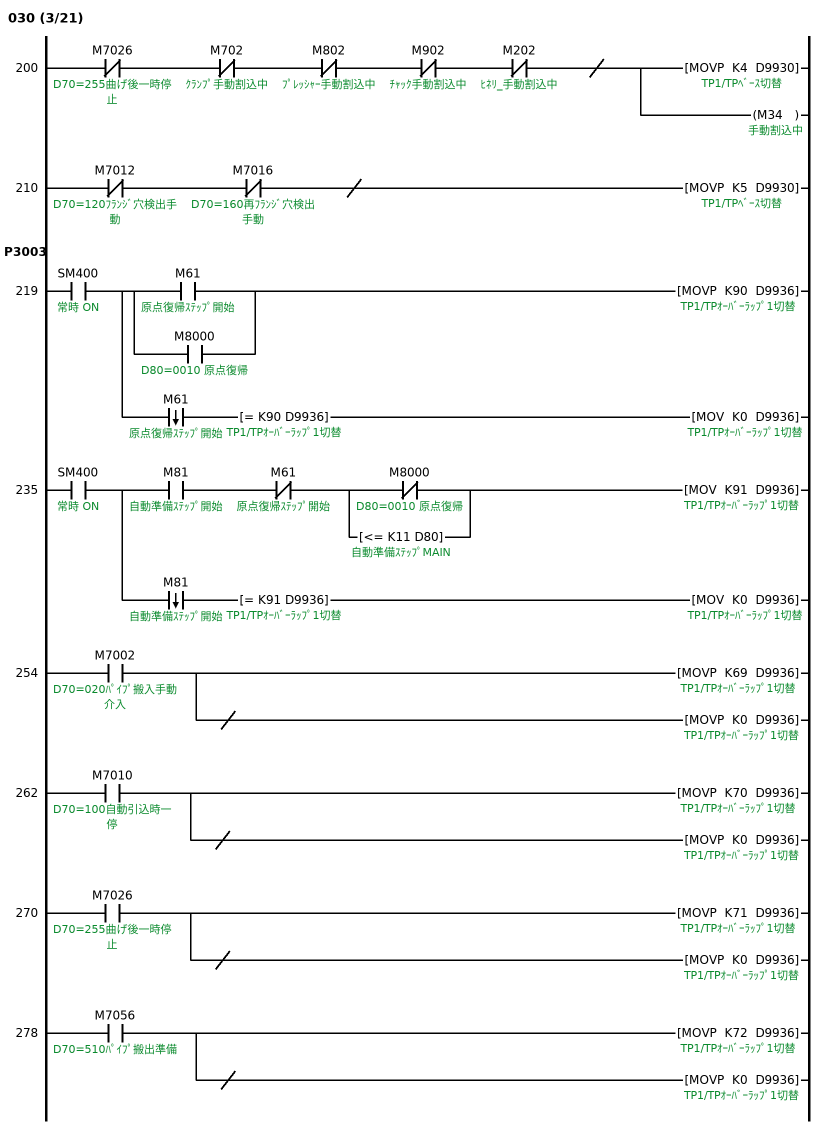
200   LDI     M7026  ; D70=255曲げ後一時停止
      ANI     M702  ; ｸﾗﾝﾌﾟ手動割込中
      ANI     M802  ; ﾌﾟﾚｯｼｬｰ手動割込中
      ANI     M902  ; ﾁｬｯｸ手動割込中
      ANI     M202  ; ﾋﾈﾘ_手動割込中
      INV
      MOVP    K4 D9930
      OUT     M34  ; 手動割込中
210   LDI     M7012  ; D70=120ﾌﾗﾝｼﾞ穴検出手動
      ANI     M7016  ; D70=160再ﾌﾗﾝｼﾞ穴検出手動
      INV
      MOVP    K5 D9930
; 
      P3003
219   LD      SM400  ; 常時 ON
      MPS
      LD      M61  ; 原点復帰ｽﾃｯﾌﾟ開始
      OR      M8000  ; D80=0010 原点復帰
      ANB
      MOVP    K90 D9936  ; TP1/TPｵｰﾊﾞｰﾗｯﾌﾟ1切替
      MPP
      ANDF    M61  ; 原点復帰ｽﾃｯﾌﾟ開始
      AND=    K90 D9936  ; TP1/TPｵｰﾊﾞｰﾗｯﾌﾟ1切替
      MOV     K0 D9936
235   LD      SM400  ; 常時 ON
      MPS
      AND     M81  ; 自動準備ｽﾃｯﾌﾟ開始
      ANI     M61  ; 原点復帰ｽﾃｯﾌﾟ開始
      LDI     M8000  ; D80=0010 原点復帰
      OR<=    K11 D80  ; 自動準備ｽﾃｯﾌﾟMAIN
      ANB
      MOV     K91 D9936
      MPP
      ANDF    M81  ; 自動準備ｽﾃｯﾌﾟ開始
      AND=    K91 D9936  ; TP1/TPｵｰﾊﾞｰﾗｯﾌﾟ1切替
      MOV     K0 D9936
254   LD      M7002  ; D70=020ﾊﾟｲﾌﾟ搬入手動介入
      MOVP    K69 D9936
      INV
      MOVP    K0 D9936
262   LD      M7010  ; D70=100自動引込時一停
      MOVP    K70 D9936
      INV
      MOVP    K0 D9936
270   LD      M7026  ; D70=255曲げ後一時停止
      MOVP    K71 D9936
      INV
      MOVP    K0 D9936
278   LD      M7056  ; D70=510ﾊﾟｲﾌﾟ搬出準備
      MOVP    K72 D9936
      INV
      MOVP    K0 D9936
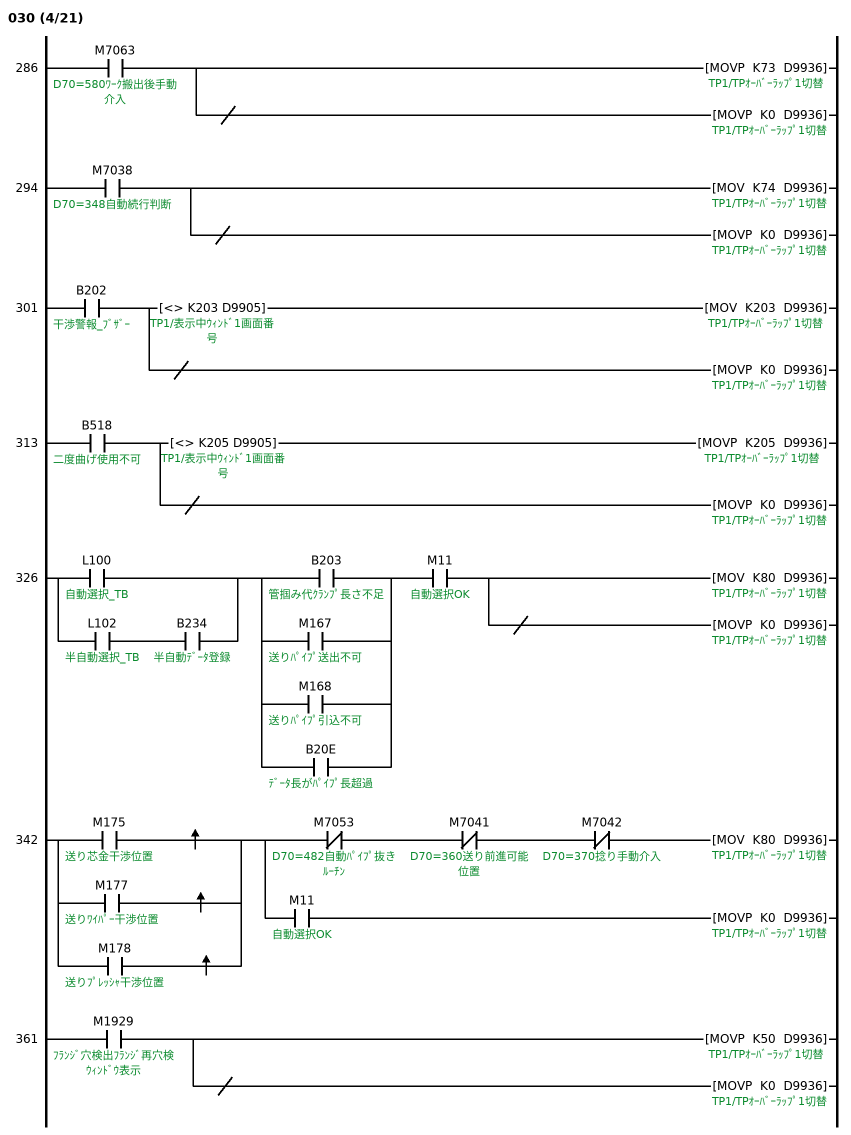
286   LD      M7063  ; D70=580ﾜｰｸ搬出後手動介入
      MOVP    K73 D9936
      INV
      MOVP    K0 D9936
294   LD      M7038  ; D70=348自動続行判断
      MOV     K74 D9936
      INV
      MOVP    K0 D9936
301   LD      B202  ; 干渉警報_ﾌﾞｻﾞｰ
      MPS
      AND<>   K203 D9905  ; TP1/表示中ｳｨﾝﾄﾞ1画面番号
      MOV     K203 D9936
      MPP
      INV
      MOVP    K0 D9936
313   LD      B518  ; 二度曲げ使用不可
      MPS
      AND<>   K205 D9905  ; TP1/表示中ｳｨﾝﾄﾞ1画面番号
      MOVP    K205 D9936
      MPP
      INV
      MOVP    K0 D9936
326   LD      L100  ; 自動選択_TB
      LD      L102  ; 半自動選択_TB
      AND     B234  ; 半自動ﾃﾞｰﾀ登録
      ORB
      LD      B203  ; 管掴み代ｸﾗﾝﾌﾟ長さ不足
      OR      M167  ; 送りﾊﾟｲﾌﾟ送出不可
      OR      M168  ; 送りﾊﾟｲﾌﾟ引込不可
      OR      B20E  ; ﾃﾞｰﾀ長がﾊﾟｲﾌﾟ長超過
      ANB
      AND     M11  ; 自動選択OK
      MOV     K80 D9936
      INV
      MOVP    K0 D9936
342   LD      M175  ; 送り芯金干渉位置
      MEP
      LD      M177  ; 送りﾜｲﾊﾟｰ干渉位置
      MEP
      ORB
      LD      M178  ; 送りﾌﾟﾚｯｼｬ干渉位置
      MEP
      ORB
      MPS
      ANI     M7053  ; D70=482自動ﾊﾟｲﾌﾟ抜きﾙｰﾁﾝ
      ANI     M7041  ; D70=360送り前進可能位置
      ANI     M7042  ; D70=370捻り手動介入
      MOV     K80 D9936
      MPP
      AND     M11  ; 自動選択OK
      MOVP    K0 D9936
361   LD      M1929  ; ﾌﾗﾝｼﾞ穴検出ﾌﾗﾝｼﾞ再穴検ｳｨﾝﾄﾞｳ表示
      MOVP    K50 D9936
      INV
      MOVP    K0 D9936
; 
      P3010
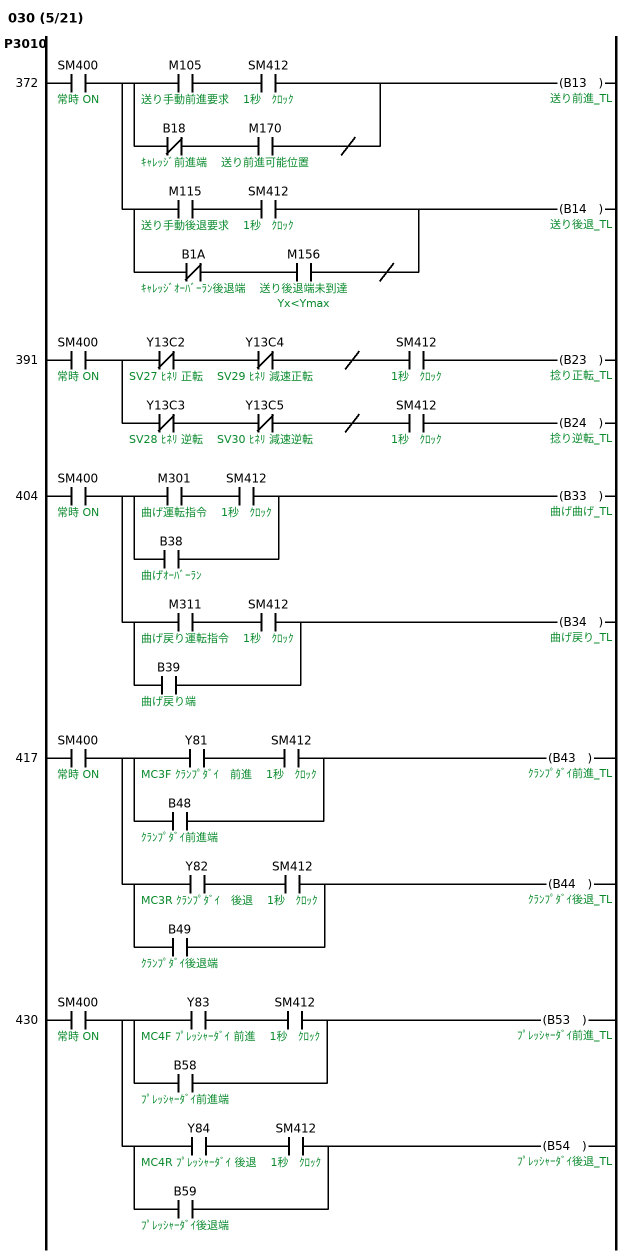
372   LD      SM400  ; 常時 ON
      MPS
      LD      M105  ; 送り手動前進要求
      AND     SM412  ; 1秒   ｸﾛｯｸ
      LDI     B18  ; ｷｬﾚｯｼﾞ前進端
      AND     M170  ; 送り前進可能位置
      INV
      ORB
      ANB
      OUT     B13  ; 送り前進_TL
      MPP
      LD      M115  ; 送り手動後退要求
      AND     SM412  ; 1秒   ｸﾛｯｸ
      LDI     B1A  ; ｷｬﾚｯｼﾞｵｰﾊﾞｰﾗﾝ後退端
      AND     M156  ; 送り後退端未到達 Yx<Ymax
      INV
      ORB
      ANB
      OUT     B14  ; 送り後退_TL
391   LD      SM400  ; 常時 ON
      MPS
      ANI     Y13C2  ; SV27 ﾋﾈﾘ 正転
      ANI     Y13C4  ; SV29 ﾋﾈﾘ 減速正転
      INV
      AND     SM412  ; 1秒   ｸﾛｯｸ
      OUT     B23  ; 捻り正転_TL
      MPP
      ANI     Y13C3  ; SV28 ﾋﾈﾘ 逆転
      ANI     Y13C5  ; SV30 ﾋﾈﾘ 減速逆転
      INV
      AND     SM412  ; 1秒   ｸﾛｯｸ
      OUT     B24  ; 捻り逆転_TL
404   LD      SM400  ; 常時 ON
      MPS
      LD      M301  ; 曲げ運転指令
      AND     SM412  ; 1秒   ｸﾛｯｸ
      OR      B38  ; 曲げｵｰﾊﾞｰﾗﾝ
      ANB
      OUT     B33  ; 曲げ曲げ_TL
      MPP
      LD      M311  ; 曲げ戻り運転指令
      AND     SM412  ; 1秒   ｸﾛｯｸ
      OR      B39  ; 曲げ戻り端
      ANB
      OUT     B34  ; 曲げ戻り_TL
417   LD      SM400  ; 常時 ON
      MPS
      LD      Y81  ; MC3F ｸﾗﾝﾌﾟﾀﾞｲ　前進
      AND     SM412  ; 1秒   ｸﾛｯｸ
      OR      B48  ; ｸﾗﾝﾌﾟﾀﾞｲ前進端
      ANB
      OUT     B43  ; ｸﾗﾝﾌﾟﾀﾞｲ前進_TL
      MPP
      LD      Y82  ; MC3R ｸﾗﾝﾌﾟﾀﾞｲ　後退
      AND     SM412  ; 1秒   ｸﾛｯｸ
      OR      B49  ; ｸﾗﾝﾌﾟﾀﾞｲ後退端
      ANB
      OUT     B44  ; ｸﾗﾝﾌﾟﾀﾞｲ後退_TL
430   LD      SM400  ; 常時 ON
      MPS
      LD      Y83  ; MC4F ﾌﾟﾚｯｼｬｰﾀﾞｲ 前進
      AND     SM412  ; 1秒   ｸﾛｯｸ
      OR      B58  ; ﾌﾟﾚｯｼｬｰﾀﾞｲ前進端
      ANB
      OUT     B53  ; ﾌﾟﾚｯｼｬｰﾀﾞｲ前進_TL
      MPP
      LD      Y84  ; MC4R ﾌﾟﾚｯｼｬｰﾀﾞｲ 後退
      AND     SM412  ; 1秒   ｸﾛｯｸ
      OR      B59  ; ﾌﾟﾚｯｼｬｰﾀﾞｲ後退端
      ANB
      OUT     B54  ; ﾌﾟﾚｯｼｬｰﾀﾞｲ後退_TL
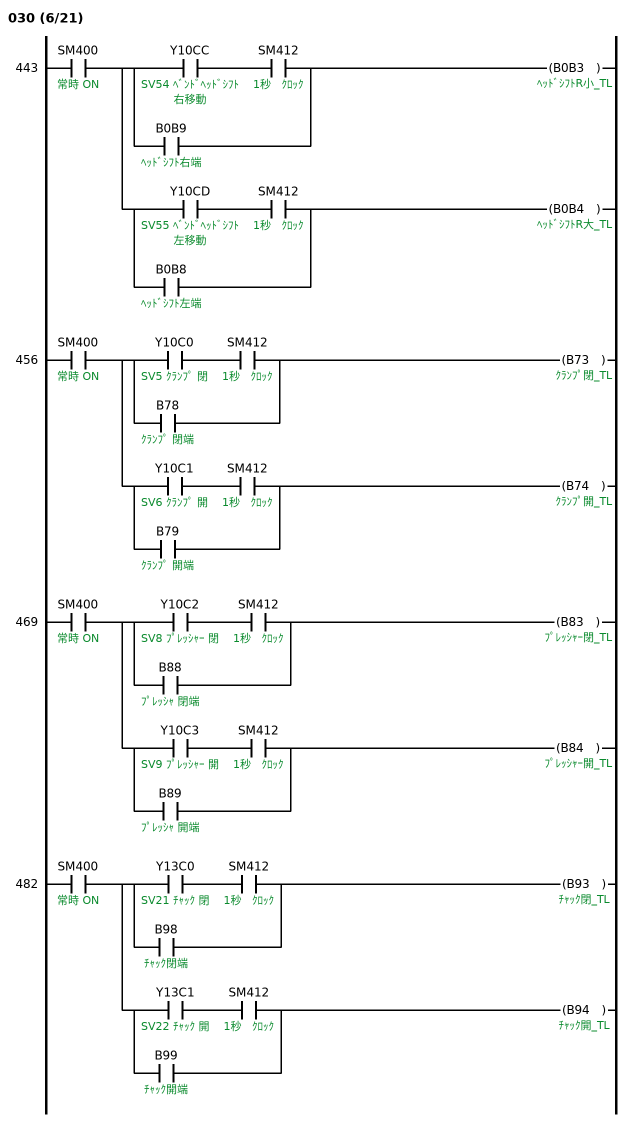
443   LD      SM400  ; 常時 ON
      MPS
      LD      Y10CC  ; SV54 ﾍﾞﾝﾄﾞﾍｯﾄﾞｼﾌﾄ 右移動
      AND     SM412  ; 1秒   ｸﾛｯｸ
      OR      B0B9  ; ﾍｯﾄﾞｼﾌﾄ右端
      ANB
      OUT     B0B3  ; ﾍｯﾄﾞｼﾌﾄR小_TL
      MPP
      LD      Y10CD  ; SV55 ﾍﾞﾝﾄﾞﾍｯﾄﾞｼﾌﾄ 左移動
      AND     SM412  ; 1秒   ｸﾛｯｸ
      OR      B0B8  ; ﾍｯﾄﾞｼﾌﾄ左端
      ANB
      OUT     B0B4  ; ﾍｯﾄﾞｼﾌﾄR大_TL
456   LD      SM400  ; 常時 ON
      MPS
      LD      Y10C0  ; SV5 ｸﾗﾝﾌﾟ 閉
      AND     SM412  ; 1秒   ｸﾛｯｸ
      OR      B78  ; ｸﾗﾝﾌﾟ 閉端
      ANB
      OUT     B73  ; ｸﾗﾝﾌﾟ閉_TL
      MPP
      LD      Y10C1  ; SV6 ｸﾗﾝﾌﾟ 開
      AND     SM412  ; 1秒   ｸﾛｯｸ
      OR      B79  ; ｸﾗﾝﾌﾟ 開端
      ANB
      OUT     B74  ; ｸﾗﾝﾌﾟ開_TL
469   LD      SM400  ; 常時 ON
      MPS
      LD      Y10C2  ; SV8 ﾌﾟﾚｯｼｬｰ 閉
      AND     SM412  ; 1秒   ｸﾛｯｸ
      OR      B88  ; ﾌﾟﾚｯｼｬ 閉端
      ANB
      OUT     B83  ; ﾌﾟﾚｯｼｬｰ閉_TL
      MPP
      LD      Y10C3  ; SV9 ﾌﾟﾚｯｼｬｰ 開
      AND     SM412  ; 1秒   ｸﾛｯｸ
      OR      B89  ; ﾌﾟﾚｯｼｬ 開端
      ANB
      OUT     B84  ; ﾌﾟﾚｯｼｬｰ開_TL
482   LD      SM400  ; 常時 ON
      MPS
      LD      Y13C0  ; SV21 ﾁｬｯｸ 閉
      AND     SM412  ; 1秒   ｸﾛｯｸ
      OR      B98  ; ﾁｬｯｸ閉端
      ANB
      OUT     B93  ; ﾁｬｯｸ閉_TL
      MPP
      LD      Y13C1  ; SV22 ﾁｬｯｸ 開
      AND     SM412  ; 1秒   ｸﾛｯｸ
      OR      B99  ; ﾁｬｯｸ開端
      ANB
      OUT     B94  ; ﾁｬｯｸ開_TL
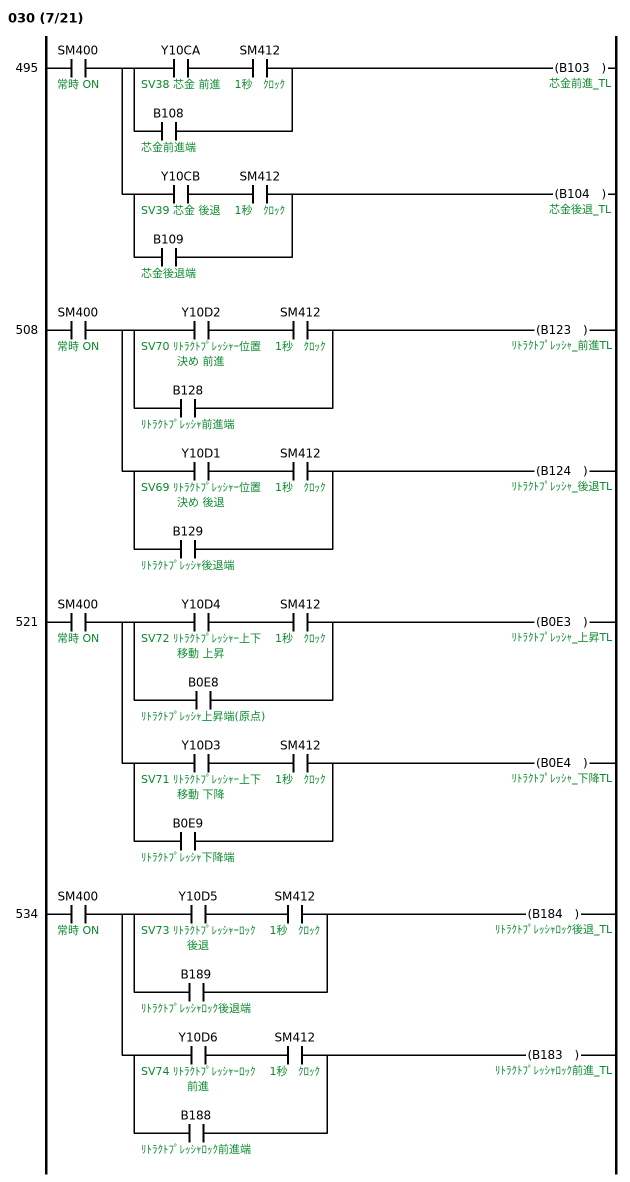
495   LD      SM400  ; 常時 ON
      MPS
      LD      Y10CA  ; SV38 芯金 前進
      AND     SM412  ; 1秒   ｸﾛｯｸ
      OR      B108  ; 芯金前進端
      ANB
      OUT     B103  ; 芯金前進_TL
      MPP
      LD      Y10CB  ; SV39 芯金 後退
      AND     SM412  ; 1秒   ｸﾛｯｸ
      OR      B109  ; 芯金後退端
      ANB
      OUT     B104  ; 芯金後退_TL
508   LD      SM400  ; 常時 ON
      MPS
      LD      Y10D2  ; SV70 ﾘﾄﾗｸﾄﾌﾟﾚｯｼｬｰ位置決め 前進
      AND     SM412  ; 1秒   ｸﾛｯｸ
      OR      B128  ; ﾘﾄﾗｸﾄﾌﾟﾚｯｼｬ前進端
      ANB
      OUT     B123  ; ﾘﾄﾗｸﾄﾌﾟﾚｯｼｬ_前進TL
      MPP
      LD      Y10D1  ; SV69 ﾘﾄﾗｸﾄﾌﾟﾚｯｼｬｰ位置決め 後退
      AND     SM412  ; 1秒   ｸﾛｯｸ
      OR      B129  ; ﾘﾄﾗｸﾄﾌﾟﾚｯｼｬ後退端
      ANB
      OUT     B124  ; ﾘﾄﾗｸﾄﾌﾟﾚｯｼｬ_後退TL
521   LD      SM400  ; 常時 ON
      MPS
      LD      Y10D4  ; SV72 ﾘﾄﾗｸﾄﾌﾟﾚｯｼｬｰ上下移動 上昇
      AND     SM412  ; 1秒   ｸﾛｯｸ
      OR      B0E8  ; ﾘﾄﾗｸﾄﾌﾟﾚｯｼｬ上昇端(原点)
      ANB
      OUT     B0E3  ; ﾘﾄﾗｸﾄﾌﾟﾚｯｼｬ_上昇TL
      MPP
      LD      Y10D3  ; SV71 ﾘﾄﾗｸﾄﾌﾟﾚｯｼｬｰ上下移動 下降
      AND     SM412  ; 1秒   ｸﾛｯｸ
      OR      B0E9  ; ﾘﾄﾗｸﾄﾌﾟﾚｯｼｬ下降端
      ANB
      OUT     B0E4  ; ﾘﾄﾗｸﾄﾌﾟﾚｯｼｬ_下降TL
534   LD      SM400  ; 常時 ON
      MPS
      LD      Y10D5  ; SV73 ﾘﾄﾗｸﾄﾌﾟﾚｯｼｬｰﾛｯｸ 後退
      AND     SM412  ; 1秒   ｸﾛｯｸ
      OR      B189  ; ﾘﾄﾗｸﾄﾌﾟﾚｯｼｬﾛｯｸ後退端
      ANB
      OUT     B184  ; ﾘﾄﾗｸﾄﾌﾟﾚｯｼｬﾛｯｸ後退_TL
      MPP
      LD      Y10D6  ; SV74 ﾘﾄﾗｸﾄﾌﾟﾚｯｼｬｰﾛｯｸ 前進
      AND     SM412  ; 1秒   ｸﾛｯｸ
      OR      B188  ; ﾘﾄﾗｸﾄﾌﾟﾚｯｼｬﾛｯｸ前進端
      ANB
      OUT     B183  ; ﾘﾄﾗｸﾄﾌﾟﾚｯｼｬﾛｯｸ前進_TL
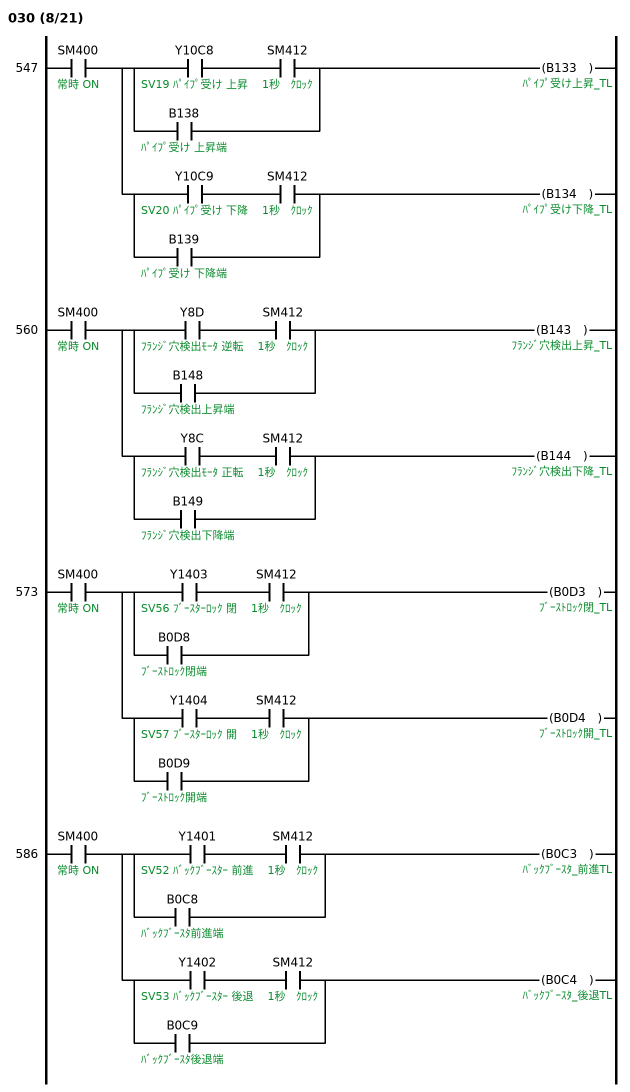
547   LD      SM400  ; 常時 ON
      MPS
      LD      Y10C8  ; SV19 ﾊﾟｲﾌﾟ受け 上昇
      AND     SM412  ; 1秒   ｸﾛｯｸ
      OR      B138  ; ﾊﾟｲﾌﾟ受け 上昇端
      ANB
      OUT     B133  ; ﾊﾟｲﾌﾟ受け上昇_TL
      MPP
      LD      Y10C9  ; SV20 ﾊﾟｲﾌﾟ受け 下降
      AND     SM412  ; 1秒   ｸﾛｯｸ
      OR      B139  ; ﾊﾟｲﾌﾟ受け 下降端
      ANB
      OUT     B134  ; ﾊﾟｲﾌﾟ受け下降_TL
560   LD      SM400  ; 常時 ON
      MPS
      LD      Y8D  ; ﾌﾗﾝｼﾞ穴検出ﾓｰﾀ 逆転
      AND     SM412  ; 1秒   ｸﾛｯｸ
      OR      B148  ; ﾌﾗﾝｼﾞ穴検出上昇端
      ANB
      OUT     B143  ; ﾌﾗﾝｼﾞ穴検出上昇_TL
      MPP
      LD      Y8C  ; ﾌﾗﾝｼﾞ穴検出ﾓｰﾀ 正転
      AND     SM412  ; 1秒   ｸﾛｯｸ
      OR      B149  ; ﾌﾗﾝｼﾞ穴検出下降端
      ANB
      OUT     B144  ; ﾌﾗﾝｼﾞ穴検出下降_TL
573   LD      SM400  ; 常時 ON
      MPS
      LD      Y1403  ; SV56 ﾌﾞｰｽﾀｰﾛｯｸ 閉
      AND     SM412  ; 1秒   ｸﾛｯｸ
      OR      B0D8  ; ﾌﾞｰｽﾄﾛｯｸ閉端
      ANB
      OUT     B0D3  ; ﾌﾞｰｽﾄﾛｯｸ閉_TL
      MPP
      LD      Y1404  ; SV57 ﾌﾞｰｽﾀｰﾛｯｸ 開
      AND     SM412  ; 1秒   ｸﾛｯｸ
      OR      B0D9  ; ﾌﾞｰｽﾄﾛｯｸ開端
      ANB
      OUT     B0D4  ; ﾌﾞｰｽﾄﾛｯｸ開_TL
586   LD      SM400  ; 常時 ON
      MPS
      LD      Y1401  ; SV52 ﾊﾞｯｸﾌﾞｰｽﾀｰ 前進
      AND     SM412  ; 1秒   ｸﾛｯｸ
      OR      B0C8  ; ﾊﾞｯｸﾌﾞｰｽﾀ前進端
      ANB
      OUT     B0C3  ; ﾊﾞｯｸﾌﾞｰｽﾀ_前進TL
      MPP
      LD      Y1402  ; SV53 ﾊﾞｯｸﾌﾞｰｽﾀｰ 後退
      AND     SM412  ; 1秒   ｸﾛｯｸ
      OR      B0C9  ; ﾊﾞｯｸﾌﾞｰｽﾀ後退端
      ANB
      OUT     B0C4  ; ﾊﾞｯｸﾌﾞｰｽﾀ_後退TL
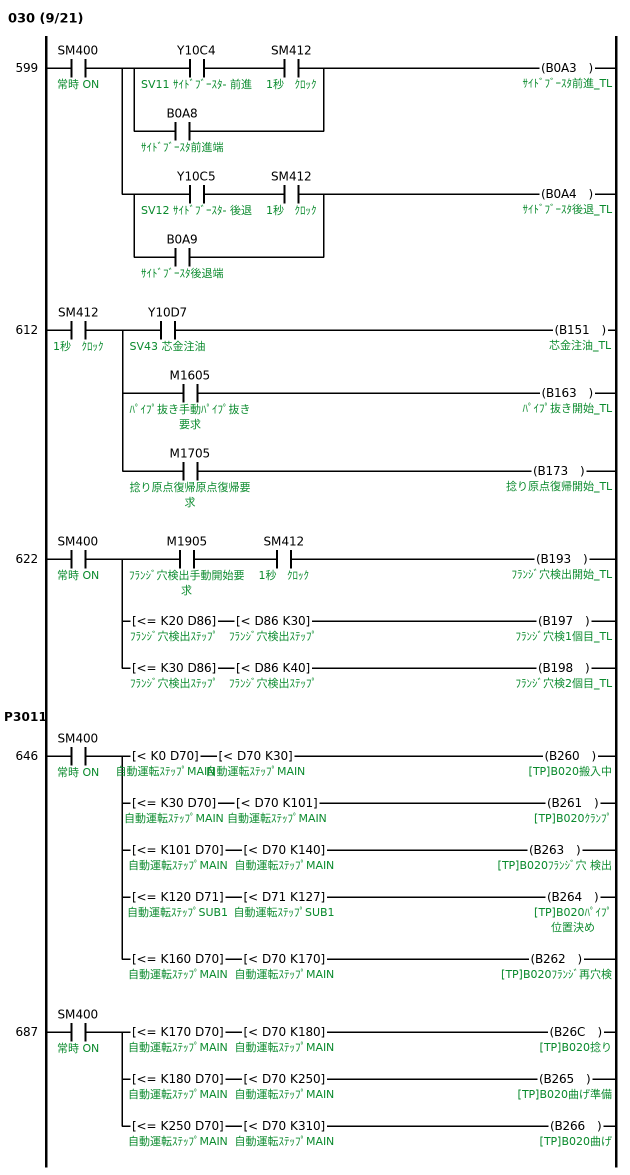
599   LD      SM400  ; 常時 ON
      MPS
      LD      Y10C4  ; SV11 ｻｲﾄﾞﾌﾞｰｽﾀ- 前進
      AND     SM412  ; 1秒   ｸﾛｯｸ
      OR      B0A8  ; ｻｲﾄﾞﾌﾞｰｽﾀ前進端
      ANB
      OUT     B0A3  ; ｻｲﾄﾞﾌﾞｰｽﾀ前進_TL
      MPP
      LD      Y10C5  ; SV12 ｻｲﾄﾞﾌﾞｰｽﾀ- 後退
      AND     SM412  ; 1秒   ｸﾛｯｸ
      OR      B0A9  ; ｻｲﾄﾞﾌﾞｰｽﾀ後退端
      ANB
      OUT     B0A4  ; ｻｲﾄﾞﾌﾞｰｽﾀ後退_TL
612   LD      SM412  ; 1秒   ｸﾛｯｸ
      MPS
      AND     Y10D7  ; SV43 芯金注油
      OUT     B151  ; 芯金注油_TL
      MRD
      AND     M1605  ; ﾊﾟｲﾌﾟ抜き手動ﾊﾟｲﾌﾟ抜き要求
      OUT     B163  ; ﾊﾟｲﾌﾟ抜き開始_TL
      MPP
      AND     M1705  ; 捻り原点復帰原点復帰要求
      OUT     B173  ; 捻り原点復帰開始_TL
622   LD      SM400  ; 常時 ON
      MPS
      AND     M1905  ; ﾌﾗﾝｼﾞ穴検出手動開始要求
      AND     SM412  ; 1秒   ｸﾛｯｸ
      OUT     B193  ; ﾌﾗﾝｼﾞ穴検出開始_TL
      MRD
      AND<=   K20 D86  ; ﾌﾗﾝｼﾞ穴検出ｽﾃｯﾌﾟ
      AND<    D86 K30  ; ﾌﾗﾝｼﾞ穴検出ｽﾃｯﾌﾟ
      OUT     B197  ; ﾌﾗﾝｼﾞ穴検1個目_TL
      MPP
      AND<=   K30 D86  ; ﾌﾗﾝｼﾞ穴検出ｽﾃｯﾌﾟ
      AND<    D86 K40  ; ﾌﾗﾝｼﾞ穴検出ｽﾃｯﾌﾟ
      OUT     B198  ; ﾌﾗﾝｼﾞ穴検2個目_TL
; 
      P3011
646   LD      SM400  ; 常時 ON
      MPS
      AND<    K0 D70  ; 自動運転ｽﾃｯﾌﾟMAIN
      AND<    D70 K30  ; 自動運転ｽﾃｯﾌﾟMAIN
      OUT     B260  ; [TP]B020搬入中
      MRD
      AND<=   K30 D70  ; 自動運転ｽﾃｯﾌﾟMAIN
      AND<    D70 K101  ; 自動運転ｽﾃｯﾌﾟMAIN
      OUT     B261  ; [TP]B020ｸﾗﾝﾌﾟ
      MRD
      AND<=   K101 D70  ; 自動運転ｽﾃｯﾌﾟMAIN
      AND<    D70 K140  ; 自動運転ｽﾃｯﾌﾟMAIN
      OUT     B263  ; [TP]B020ﾌﾗﾝｼﾞ穴 検出
      MRD
      AND<=   K120 D71  ; 自動運転ｽﾃｯﾌﾟSUB1
      AND<    D71 K127  ; 自動運転ｽﾃｯﾌﾟSUB1
      OUT     B264  ; [TP]B020ﾊﾟｲﾌﾟ   位置決め
      MPP
      AND<=   K160 D70  ; 自動運転ｽﾃｯﾌﾟMAIN
      AND<    D70 K170  ; 自動運転ｽﾃｯﾌﾟMAIN
      OUT     B262  ; [TP]B020ﾌﾗﾝｼﾞ再穴検
687   LD      SM400  ; 常時 ON
      MPS
      AND<=   K170 D70  ; 自動運転ｽﾃｯﾌﾟMAIN
      AND<    D70 K180  ; 自動運転ｽﾃｯﾌﾟMAIN
      OUT     B26C  ; [TP]B020捻り
      MRD
      AND<=   K180 D70  ; 自動運転ｽﾃｯﾌﾟMAIN
      AND<    D70 K250  ; 自動運転ｽﾃｯﾌﾟMAIN
      OUT     B265  ; [TP]B020曲げ準備
      MPP
      AND<=   K250 D70  ; 自動運転ｽﾃｯﾌﾟMAIN
      AND<    D70 K310  ; 自動運転ｽﾃｯﾌﾟMAIN
      OUT     B266  ; [TP]B020曲げ
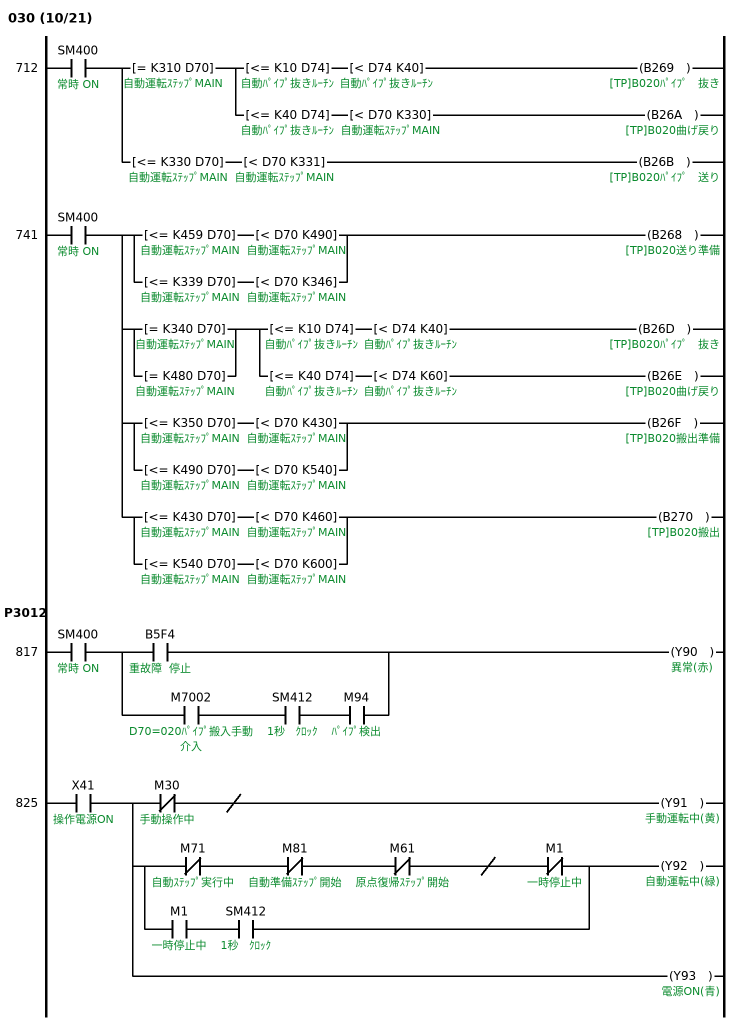
712   LD      SM400  ; 常時 ON
      MPS
      AND=    K310 D70  ; 自動運転ｽﾃｯﾌﾟMAIN
      MPS
      AND<=   K10 D74  ; 自動ﾊﾟｲﾌﾟ抜きﾙｰﾁﾝ
      AND<    D74 K40  ; 自動ﾊﾟｲﾌﾟ抜きﾙｰﾁﾝ
      OUT     B269  ; [TP]B020ﾊﾟｲﾌﾟ   抜き
      MPP
      AND<=   K40 D74  ; 自動ﾊﾟｲﾌﾟ抜きﾙｰﾁﾝ
      AND<    D70 K330  ; 自動運転ｽﾃｯﾌﾟMAIN
      OUT     B26A  ; [TP]B020曲げ戻り
      MPP
      AND<=   K330 D70  ; 自動運転ｽﾃｯﾌﾟMAIN
      AND<    D70 K331  ; 自動運転ｽﾃｯﾌﾟMAIN
      OUT     B26B  ; [TP]B020ﾊﾟｲﾌﾟ   送り
741   LD      SM400  ; 常時 ON
      MPS
      LD<=    K459 D70  ; 自動運転ｽﾃｯﾌﾟMAIN
      AND<    D70 K490  ; 自動運転ｽﾃｯﾌﾟMAIN
      LD<=    K339 D70  ; 自動運転ｽﾃｯﾌﾟMAIN
      AND<    D70 K346  ; 自動運転ｽﾃｯﾌﾟMAIN
      ORB
      ANB
      OUT     B268  ; [TP]B020送り準備
      MRD
      LD=     K340 D70  ; 自動運転ｽﾃｯﾌﾟMAIN
      OR=     K480 D70  ; 自動運転ｽﾃｯﾌﾟMAIN
      ANB
      MPS
      AND<=   K10 D74  ; 自動ﾊﾟｲﾌﾟ抜きﾙｰﾁﾝ
      AND<    D74 K40  ; 自動ﾊﾟｲﾌﾟ抜きﾙｰﾁﾝ
      OUT     B26D  ; [TP]B020ﾊﾟｲﾌﾟ   抜き
      MPP
      AND<=   K40 D74  ; 自動ﾊﾟｲﾌﾟ抜きﾙｰﾁﾝ
      AND<    D74 K60  ; 自動ﾊﾟｲﾌﾟ抜きﾙｰﾁﾝ
      OUT     B26E  ; [TP]B020曲げ戻り
      MRD
      LD<=    K350 D70  ; 自動運転ｽﾃｯﾌﾟMAIN
      AND<    D70 K430  ; 自動運転ｽﾃｯﾌﾟMAIN
      LD<=    K490 D70  ; 自動運転ｽﾃｯﾌﾟMAIN
      AND<    D70 K540  ; 自動運転ｽﾃｯﾌﾟMAIN
      ORB
      ANB
      OUT     B26F  ; [TP]B020搬出準備
      MPP
      LD<=    K430 D70  ; 自動運転ｽﾃｯﾌﾟMAIN
      AND<    D70 K460  ; 自動運転ｽﾃｯﾌﾟMAIN
      LD<=    K540 D70  ; 自動運転ｽﾃｯﾌﾟMAIN
      AND<    D70 K600  ; 自動運転ｽﾃｯﾌﾟMAIN
      ORB
      ANB
      OUT     B270  ; [TP]B020搬出
; 
      P3012
817   LD      SM400  ; 常時 ON
      LD      B5F4  ; 重故障  停止
      LD      M7002  ; D70=020ﾊﾟｲﾌﾟ搬入手動介入
      AND     SM412  ; 1秒   ｸﾛｯｸ
      AND     M94  ; ﾊﾟｲﾌﾟ検出
      ORB
      ANB
      OUT     Y90  ; 異常(赤)
825   LD      X41  ; 操作電源ON
      MPS
      ANI     M30  ; 手動操作中
      INV
      OUT     Y91  ; 手動運転中(黄)
      MRD
      LDI     M71  ; 自動ｽﾃｯﾌﾟ実行中
      ANI     M81  ; 自動準備ｽﾃｯﾌﾟ開始
      ANI     M61  ; 原点復帰ｽﾃｯﾌﾟ開始
      INV
      ANI     M1  ; 一時停止中
      LD      M1  ; 一時停止中
      AND     SM412  ; 1秒   ｸﾛｯｸ
      ORB
      ANB
      OUT     Y92  ; 自動運転中(緑)
      MPP
      OUT     Y93  ; 電源ON(青)
; 
      P3013
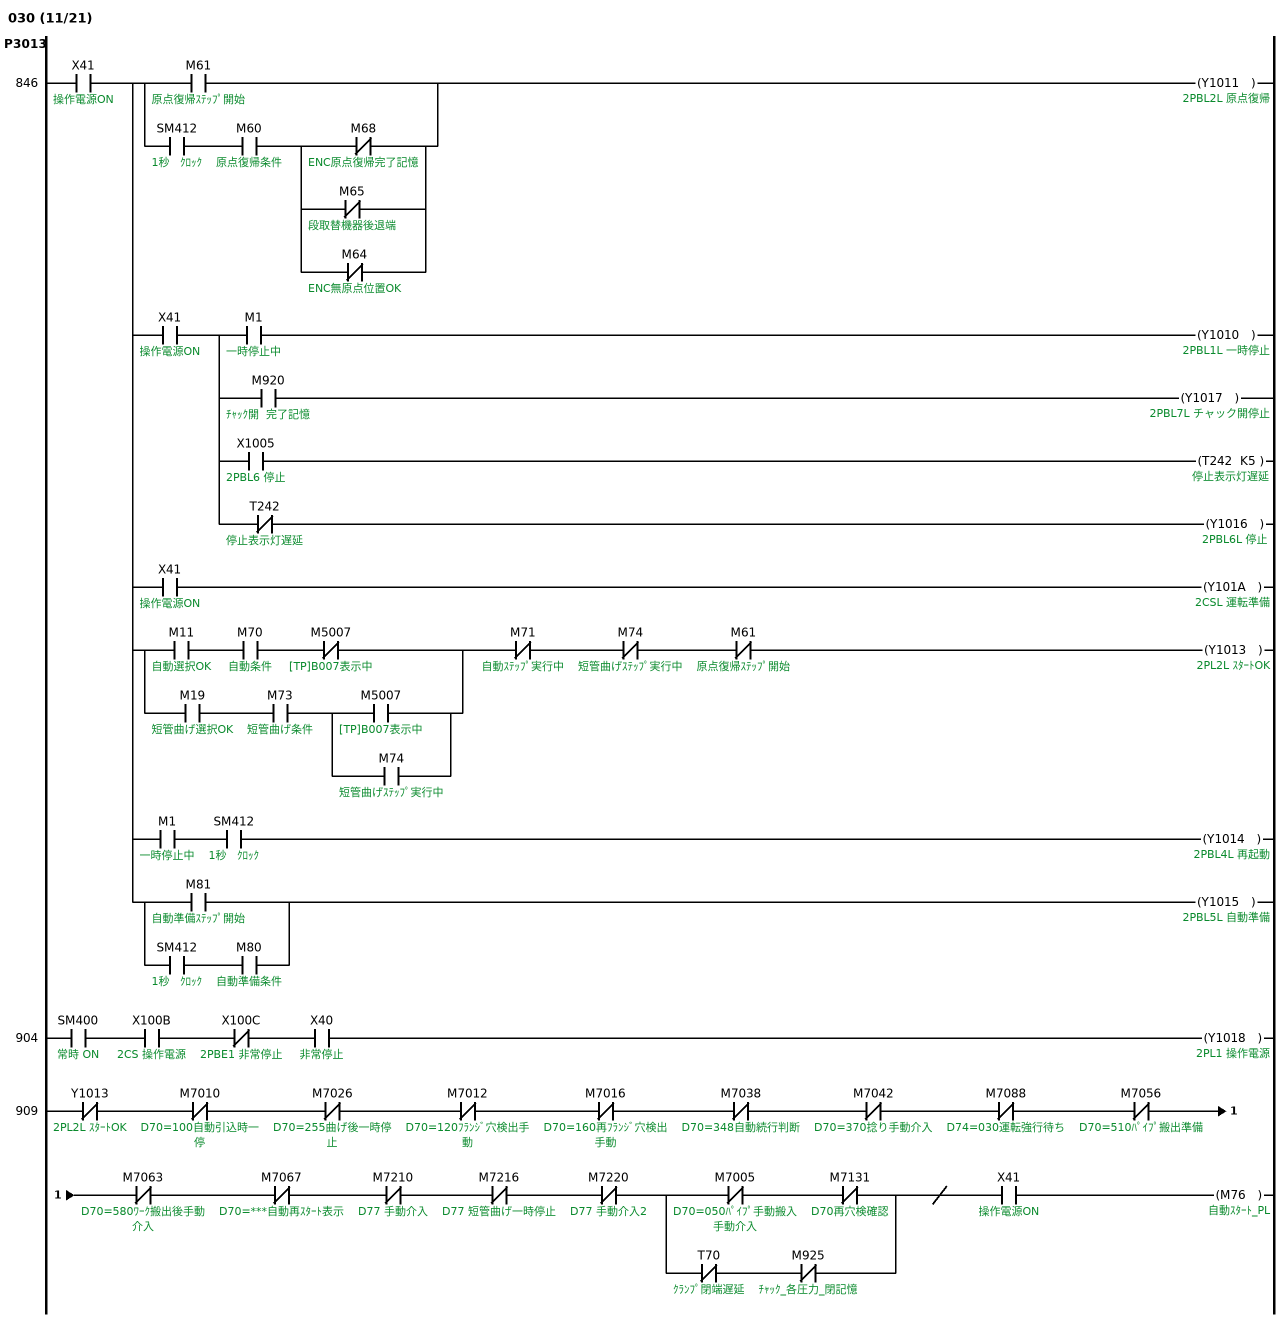
846   LD      X41  ; 操作電源ON
      MPS
      LD      M61  ; 原点復帰ｽﾃｯﾌﾟ開始
      LD      SM412  ; 1秒   ｸﾛｯｸ
      AND     M60  ; 原点復帰条件
      LDI     M68  ; ENC原点復帰完了記憶
      ORI     M65  ; 段取替機器後退端
      ORI     M64  ; ENC無原点位置OK
      ANB
      ORB
      ANB
      OUT     Y1011  ; 2PBL2L 原点復帰
      MRD
      AND     X41  ; 操作電源ON
      MPS
      AND     M1  ; 一時停止中
      OUT     Y1010  ; 2PBL1L 一時停止
      MRD
      AND     M920  ; ﾁｬｯｸ開  完了記憶
      OUT     Y1017  ; 2PBL7L チャック開停止
      MRD
      AND     X1005  ; 2PBL6 停止
      OUT     T242 K5  ; 停止表示灯遅延
      MPP
      ANI     T242  ; 停止表示灯遅延
      OUT     Y1016  ; 2PBL6L 停止
      MRD
      AND     X41  ; 操作電源ON
      OUT     Y101A  ; 2CSL 運転準備
      MRD
      LD      M11  ; 自動選択OK
      AND     M70  ; 自動条件
      ANI     M5007  ; [TP]B007表示中
      LD      M19  ; 短管曲げ選択OK
      AND     M73  ; 短管曲げ条件
      LD      M5007  ; [TP]B007表示中
      OR      M74  ; 短管曲げｽﾃｯﾌﾟ実行中
      ANB
      ORB
      ANB
      ANI     M71  ; 自動ｽﾃｯﾌﾟ実行中
      ANI     M74  ; 短管曲げｽﾃｯﾌﾟ実行中
      ANI     M61  ; 原点復帰ｽﾃｯﾌﾟ開始
      OUT     Y1013  ; 2PL2L ｽﾀｰﾄOK
      MRD
      AND     M1  ; 一時停止中
      AND     SM412  ; 1秒   ｸﾛｯｸ
      OUT     Y1014  ; 2PBL4L 再起動
      MPP
      LD      M81  ; 自動準備ｽﾃｯﾌﾟ開始
      LD      SM412  ; 1秒   ｸﾛｯｸ
      AND     M80  ; 自動準備条件
      ORB
      ANB
      OUT     Y1015  ; 2PBL5L 自動準備
904   LD      SM400  ; 常時 ON
      AND     X100B  ; 2CS 操作電源
      ANI     X100C  ; 2PBE1 非常停止
      AND     X40  ; 非常停止
      OUT     Y1018  ; 2PL1 操作電源
909   LDI     Y1013  ; 2PL2L ｽﾀｰﾄOK
      ANI     M7010  ; D70=100自動引込時一停
      ANI     M7026  ; D70=255曲げ後一時停止
      ANI     M7012  ; D70=120ﾌﾗﾝｼﾞ穴検出手動
      ANI     M7016  ; D70=160再ﾌﾗﾝｼﾞ穴検出手動
      ANI     M7038  ; D70=348自動続行判断
      ANI     M7042  ; D70=370捻り手動介入
      ANI     M7088  ; D74=030運転強行待ち
      ANI     M7056  ; D70=510ﾊﾟｲﾌﾟ搬出準備
      ANI     M7063  ; D70=580ﾜｰｸ搬出後手動介入
      ANI     M7067  ; D70=***自動再ｽﾀｰﾄ表示
      ANI     M7210  ; D77 手動介入
      ANI     M7216  ; D77 短管曲げ一時停止
      ANI     M7220  ; D77 手動介入2
      LDI     M7005  ; D70=050ﾊﾟｲﾌﾟ手動搬入手動介入
      ANI     M7131  ; D70再穴検確認
      LDI     T70  ; ｸﾗﾝﾌﾟ閉端遅延
      ANI     M925  ; ﾁｬｯｸ_各圧力_閉記憶
      ORB
      ANB
      INV
      AND     X41  ; 操作電源ON
      OUT     M76  ; 自動ｽﾀｰﾄ_PL
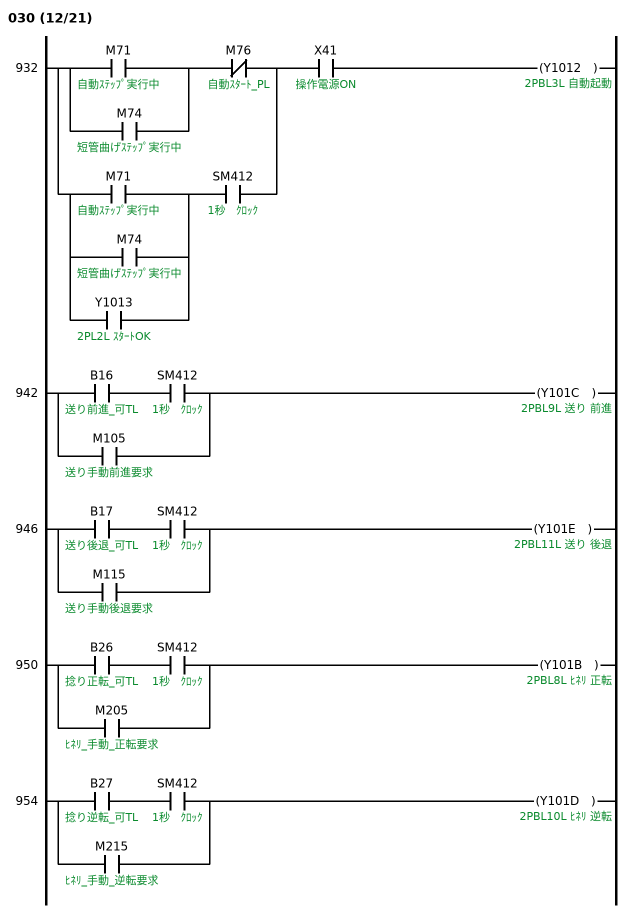
932   LD      M71  ; 自動ｽﾃｯﾌﾟ実行中
      OR      M74  ; 短管曲げｽﾃｯﾌﾟ実行中
      ANI     M76  ; 自動ｽﾀｰﾄ_PL
      LD      M71  ; 自動ｽﾃｯﾌﾟ実行中
      OR      M74  ; 短管曲げｽﾃｯﾌﾟ実行中
      OR      Y1013  ; 2PL2L ｽﾀｰﾄOK
      AND     SM412  ; 1秒   ｸﾛｯｸ
      ORB
      AND     X41  ; 操作電源ON
      OUT     Y1012  ; 2PBL3L 自動起動
942   LD      B16  ; 送り前進_可TL
      AND     SM412  ; 1秒   ｸﾛｯｸ
      OR      M105  ; 送り手動前進要求
      OUT     Y101C  ; 2PBL9L 送り 前進
946   LD      B17  ; 送り後退_可TL
      AND     SM412  ; 1秒   ｸﾛｯｸ
      OR      M115  ; 送り手動後退要求
      OUT     Y101E  ; 2PBL11L 送り 後退
950   LD      B26  ; 捻り正転_可TL
      AND     SM412  ; 1秒   ｸﾛｯｸ
      OR      M205  ; ﾋﾈﾘ_手動_正転要求
      OUT     Y101B  ; 2PBL8L ﾋﾈﾘ 正転
954   LD      B27  ; 捻り逆転_可TL
      AND     SM412  ; 1秒   ｸﾛｯｸ
      OR      M215  ; ﾋﾈﾘ_手動_逆転要求
      OUT     Y101D  ; 2PBL10L ﾋﾈﾘ 逆転
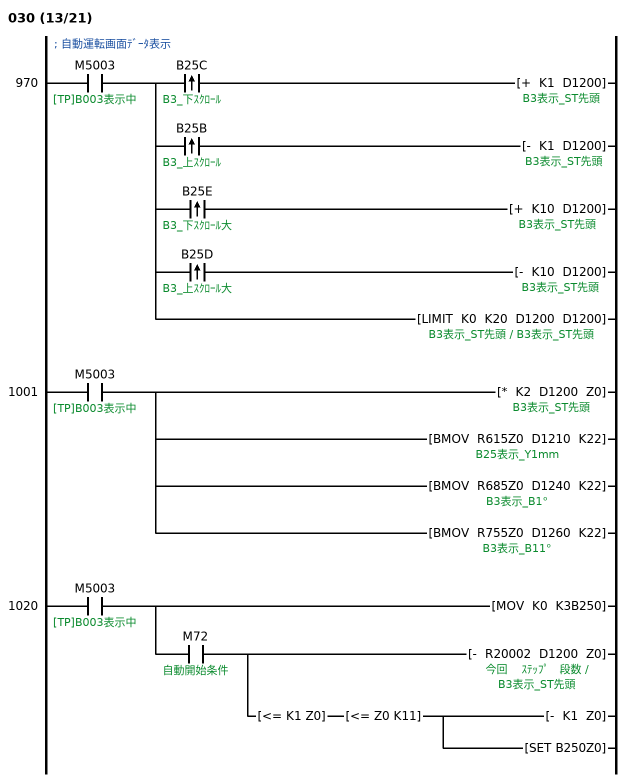
; 自動運転画面ﾃﾞｰﾀ表示
970   LD      M5003  ; [TP]B003表示中
      MPS
      ANDP    B25C  ; B3_下ｽｸﾛｰﾙ
      +       K1 D1200  ; B3表示_ST先頭
      MRD
      ANDP    B25B  ; B3_上ｽｸﾛｰﾙ
      -       K1 D1200
      MRD
      ANDP    B25E  ; B3_下ｽｸﾛｰﾙ大
      +       K10 D1200
      MRD
      ANDP    B25D  ; B3_上ｽｸﾛｰﾙ大
      -       K10 D1200
      MPP
      LIMIT   K0 K20 D1200 D1200
1001  LD      M5003  ; [TP]B003表示中
      *       K2 D1200 Z0
      BMOV    R615Z0 D1210 K22  ; B25表示_Y1mm
      BMOV    R685Z0 D1240 K22  ; B3表示_B1°
      BMOV    R755Z0 D1260 K22  ; B3表示_B11°
1020  LD      M5003  ; [TP]B003表示中
      MOV     K0 K3B250  ; B3_ST01点滅
      AND     M72  ; 自動開始条件
      -       R20002 D1200 Z0  ; 今回    ｽﾃｯﾌﾟ   段数
      AND<=   K1 Z0
      AND<=   Z0 K11
      -       K1 Z0
      SET     B250Z0
